LIN {X -0.028,Y -654.223,Z 1397.377,A 0.000,B 0.000,C 90.000,E1 103.772} C_DIS
LIN {X 0.258,Y -654.765,Z 1397.372,A 0.000,B 0.000,C 90.000,E1 103.008} C_DIS
LIN {X -0.090,Y -654.690,Z 1397.368,A 0.000,B 0.000,C 90.000,E1 102.299} C_DIS
LIN {X 0.196,Y -654.215,Z 1397.364,A 0.000,B 0.000,C 90.000,E1 101.535} C_DIS
LIN {X -0.172,Y -653.704,Z 1397.361,A 0.000,B 0.000,C 90.000,E1 101.074} C_DIS
LIN {X 0.100,Y -652.649,Z 1397.357,A 0.000,B 0.000,C 90.000,E1 100.310} C_DIS
LIN {X -0.269,Y -651.574,Z 1397.355,A 0.000,B 0.000,C 90.000,E1 99.849} C_DIS
LIN {X -0.133,Y -649.621,Z 1397.350,A 0.000,B 0.000,C 90.000,E1 99.095} C_DIS
LIN {X 0.226,Y -648.028,Z 1397.348,A 0.000,B 0.000,C 90.000,E1 98.568} C_DIS
LIN {X 0.320,Y -645.227,Z 1397.344,A 0.000,B 0.000,C 90.000,E1 97.814} C_DIS
LIN {X -0.334,Y -641.988,Z 1397.339,A 0.000,B 0.000,C 90.000,E1 97.125} C_DIS
LIN {X 0.006,Y -640.157,Z 1397.337,A 0.000,B 0.000,C 90.000,E1 96.720} C_DIS
LIN {X -0.120,Y -635.379,Z 1397.333,A 0.000,B 0.000,C 90.000,E1 95.853} C_DIS
LIN {X -0.229,Y -630.892,Z 1397.328,A 0.000,B 0.000,C 90.000,E1 95.106} C_DIS
LIN {X 0.039,Y -628.510,Z 1397.326,A 0.000,B 0.000,C 90.000,E1 94.702} C_DIS
LIN {X -0.040,Y -623.882,Z 1397.323,A 0.000,B 0.000,C 90.000,E1 94.073} C_DIS
LIN {X 0.039,Y -619.403,Z 1397.320,A 0.000,B 0.000,C 90.000,E1 93.555} C_DIS
LIN {X 0.122,Y -612.923,Z 1397.316,A 0.000,B 0.000,C 90.000,E1 92.922} C_DIS
LIN {X -0.217,Y -603.430,Z 1397.312,A 0.000,B 0.000,C 90.000,E1 92.121} C_DIS
LIN {X -0.253,Y -596.324,Z 1397.308,A 0.000,B 0.000,C 90.000,E1 91.547} C_DIS
LIN {X 0.108,Y -590.137,Z 1397.306,A 0.000,B 0.000,C 90.000,E1 91.088} C_DIS
LIN {X 0.184,Y -581.549,Z 1397.304,A 0.000,B 0.000,C 90.000,E1 90.630} C_DIS
LIN {X 0.247,Y -578.421,Z 1397.303,A 0.000,B 0.000,C 90.000,E1 90.458} C_DIS
LIN {X -0.091,Y -574.450,Z 1397.301,A 0.000,B 0.000,C 90.000,E1 90.172} C_DIS
LIN {X -0.127,Y -574.415,Z 1397.301,A 0.000,B 0.000,C 90.000,E1 90.172} C_DIS
LIN {X 0.227,Y -574.050,Z 1397.301,A 0.000,B 0.000,C 90.000,E1 90.057} C_DIS
LIN {X -0.012,Y -573.513,Z 1397.299,A 0.000,B 0.000,C 90.000,E1 89.828} C_DIS
LIN {X -0.202,Y -573.490,Z 1397.296,A 0.000,B 0.000,C 90.000,E1 89.370} C_DIS
LIN {X 0.249,Y -575.095,Z 1397.286,A 0.000,B 0.000,C 90.000,E1 87.421} C_DIS
LIN {X -0.237,Y -577.045,Z 1397.274,A 0.000,B 0.000,C 90.000,E1 85.298} C_DIS
LIN {X -0.145,Y -579.107,Z 1397.263,A 0.000,B 0.000,C 90.000,E1 83.394} C_DIS
LIN {X 0.007,Y -581.279,Z 1397.253,A 0.000,B 0.000,C 90.000,E1 81.489} C_DIS
LIN {X 0.257,Y -582.556,Z 1397.247,A 0.000,B 0.000,C 90.000,E1 80.387} C_DIS
LIN {X -0.052,Y -583.764,Z 1397.241,A 0.000,B 0.000,C 90.000,E1 79.342} C_DIS
LIN {X -0.236,Y -584.942,Z 1397.235,A 0.000,B 0.000,C 90.000,E1 78.285} C_DIS
LIN {X 0.094,Y -586.345,Z 1397.226,A 0.000,B 0.000,C 90.000,E1 76.645} C_DIS
LIN {X 0.019,Y -587.620,Z 1397.217,A 0.000,B 0.000,C 90.000,E1 75.046} C_DIS
LIN {X -0.040,Y -588.586,Z 1397.208,A 0.000,B 0.000,C 90.000,E1 73.449} C_DIS
LIN {X -0.063,Y -589.644,Z 1397.198,A 0.000,B 0.000,C 90.000,E1 71.583} C_DIS
LIN {X -0.302,Y -590.537,Z 1397.189,A 0.000,B 0.000,C 90.000,E1 70.007} C_DIS
LIN {X -0.097,Y -591.958,Z 1397.176,A 0.000,B 0.000,C 90.000,E1 67.592} C_DIS
LIN {X -0.192,Y -593.241,Z 1397.165,A 0.000,B 0.000,C 90.000,E1 65.741} C_DIS
LIN {X 0.124,Y -594.937,Z 1397.153,A 0.000,B 0.000,C 90.000,E1 63.589} C_DIS
LIN {X -0.049,Y -595.962,Z 1397.146,A 0.000,B 0.000,C 90.000,E1 62.281} C_DIS
LIN {X 0.329,Y -597.051,Z 1397.139,A 0.000,B 0.000,C 90.000,E1 60.923} C_DIS
LIN {X 0.281,Y -598.053,Z 1397.133,A 0.000,B 0.000,C 90.000,E1 59.871} C_DIS
LIN {X -0.130,Y -599.514,Z 1397.124,A 0.000,B 0.000,C 90.000,E1 58.329} C_DIS
LIN {X 0.074,Y -600.723,Z 1397.117,A 0.000,B 0.000,C 90.000,E1 56.993} C_DIS
LIN {X -0.126,Y -601.706,Z 1397.111,A 0.000,B 0.000,C 90.000,E1 55.960} C_DIS
LIN {X -0.049,Y -603.347,Z 1397.101,A 0.000,B 0.000,C 90.000,E1 54.116} C_DIS
LIN {X -0.187,Y -604.711,Z 1397.092,A 0.000,B 0.000,C 90.000,E1 52.557} C_DIS
LIN {X -0.201,Y -605.659,Z 1397.085,A 0.000,B 0.000,C 90.000,E1 51.251} C_DIS
LIN {X -0.084,Y -606.259,Z 1397.079,A 0.000,B 0.000,C 90.000,E1 50.194} C_DIS
LIN {X 0.047,Y -606.765,Z 1397.073,A 0.000,B 0.000,C 90.000,E1 49.138} C_DIS
LIN {X 0.250,Y -607.155,Z 1397.064,A 0.000,B 0.000,C 90.000,E1 47.553} C_DIS
LIN {X -0.255,Y -607.255,Z 1397.057,A 0.000,B 0.000,C 90.000,E1 46.296} C_DIS
LIN {X -0.337,Y -607.136,Z 1397.050,A 0.000,B 0.000,C 90.000,E1 45.000} C_DIS
LIN {X -0.230,Y -606.904,Z 1397.044,A 0.000,B 0.000,C 90.000,E1 43.947} C_DIS
LIN {X 0.117,Y -606.327,Z 1397.037,A 0.000,B 0.000,C 90.000,E1 42.609} C_DIS
LIN {X -0.211,Y -605.753,Z 1397.031,A 0.000,B 0.000,C 90.000,E1 41.595} C_DIS
LIN {X 0.165,Y -604.895,Z 1397.024,A 0.000,B 0.000,C 90.000,E1 40.253} C_DIS
LIN {X 0.013,Y -604.259,Z 1397.019,A 0.000,B 0.000,C 90.000,E1 39.483} C_DIS
LIN {X -0.019,Y -602.878,Z 1397.012,A 0.000,B 0.000,C 90.000,E1 38.177} C_DIS
LIN {X 0.269,Y -601.993,Z 1397.008,A 0.000,B 0.000,C 90.000,E1 37.363} C_DIS
LIN {X -0.164,Y -600.049,Z 1397.000,A 0.000,B 0.000,C 90.000,E1 36.091} C_DIS
LIN {X -0.270,Y -598.638,Z 1396.996,A 0.000,B 0.000,C 90.000,E1 35.311} C_DIS
LIN {X 0.101,Y -597.046,Z 1396.992,A 0.000,B 0.000,C 90.000,E1 34.485} C_DIS
LIN {X 0.077,Y -594.080,Z 1396.984,A 0.000,B 0.000,C 90.000,E1 33.166} C_DIS
LIN {X 0.395,Y -592.041,Z 1396.980,A 0.000,B 0.000,C 90.000,E1 32.339} C_DIS
LIN {X -0.240,Y -588.887,Z 1396.974,A 0.000,B 0.000,C 90.000,E1 31.337} C_DIS
LIN {X -0.167,Y -587.077,Z 1396.971,A 0.000,B 0.000,C 90.000,E1 30.797} C_DIS
LIN {X -0.231,Y -584.064,Z 1396.967,A 0.000,B 0.000,C 90.000,E1 30.001} C_DIS
LIN {X 0.179,Y -580.561,Z 1396.962,A 0.000,B 0.000,C 90.000,E1 29.155} C_DIS
LIN {X 0.187,Y -578.017,Z 1396.959,A 0.000,B 0.000,C 90.000,E1 28.615} C_DIS
LIN {X -0.180,Y -574.660,Z 1396.955,A 0.000,B 0.000,C 90.000,E1 27.975} C_DIS
LIN {X 0.120,Y -570.350,Z 1396.951,A 0.000,B 0.000,C 90.000,E1 27.129} C_DIS
LIN {X 0.114,Y -565.642,Z 1396.946,A 0.000,B 0.000,C 90.000,E1 26.309} C_DIS
LIN {X 0.305,Y -560.595,Z 1396.942,A 0.000,B 0.000,C 90.000,E1 25.463} C_DIS
LIN {X 0.303,Y -556.030,Z 1396.938,A 0.000,B 0.000,C 90.000,E1 24.771} C_DIS
LIN {X 0.146,Y -550.011,Z 1396.933,A 0.000,B 0.000,C 90.000,E1 23.951} C_DIS
LIN {X 0.049,Y -544.578,Z 1396.929,A 0.000,B 0.000,C 90.000,E1 23.259} C_DIS
LIN {X 0.060,Y -537.580,Z 1396.925,A 0.000,B 0.000,C 90.000,E1 22.408} C_DIS
LIN {X 0.026,Y -531.509,Z 1396.921,A 0.000,B 0.000,C 90.000,E1 21.716} C_DIS
LIN {X 0.295,Y -525.047,Z 1396.917,A 0.000,B 0.000,C 90.000,E1 20.972} C_DIS
LIN {X 0.144,Y -515.882,Z 1396.911,A 0.000,B 0.000,C 90.000,E1 19.993} C_DIS
LIN {X -0.024,Y -510.423,Z 1396.908,A 0.000,B 0.000,C 90.000,E1 19.450} C_DIS
LIN {X -0.067,Y -500.976,Z 1396.903,A 0.000,B 0.000,C 90.000,E1 18.489} C_DIS
LIN {X -0.077,Y -493.128,Z 1396.898,A 0.000,B 0.000,C 90.000,E1 17.692} C_DIS
LIN {X -0.209,Y -479.603,Z 1396.891,A 0.000,B 0.000,C 90.000,E1 16.315} C_DIS
LIN {X -0.202,Y -463.211,Z 1396.881,A 0.000,B 0.000,C 90.000,E1 14.592} C_DIS
LIN {X 0.213,Y -449.337,Z 1396.873,A 0.000,B 0.000,C 90.000,E1 13.063} C_DIS
LIN {X -0.042,Y -438.331,Z 1396.866,A 0.000,B 0.000,C 90.000,E1 11.883} C_DIS
LIN {X 0.139,Y -428.813,Z 1396.860,A 0.000,B 0.000,C 90.000,E1 10.782} C_DIS
LIN {X -0.148,Y -412.657,Z 1396.849,A 0.000,B 0.000,C 90.000,E1 8.859} C_DIS
LIN {X 0.054,Y -401.725,Z 1396.842,A 0.000,B 0.000,C 90.000,E1 7.466} C_DIS
LIN {X 0.139,Y -392.488,Z 1396.835,A 0.000,B 0.000,C 90.000,E1 6.258} C_DIS
LIN {X -0.029,Y -389.440,Z 1396.832,A 0.000,B 0.000,C 90.000,E1 5.796} C_DIS
LIN {X -0.162,Y -389.042,Z 1396.832,A 0.000,B 0.000,C 90.000,E1 5.682} C_DIS
LIN {X 0.188,Y -389.043,Z 1396.831,A 0.000,B 0.000,C 90.000,E1 5.625} C_DIS
LIN {X -0.051,Y -389.537,Z 1396.830,A 0.000,B 0.000,C 90.000,E1 5.454} C_DIS
LIN {X -0.089,Y -389.567,Z 1396.830,A 0.000,B 0.000,C 90.000,E1 5.454} C_DIS
LIN {X 0.043,Y -392.874,Z 1396.828,A 0.000,B 0.000,C 90.000,E1 5.049} C_DIS
LIN {X 0.057,Y -404.273,Z 1396.822,A 0.000,B 0.000,C 90.000,E1 4.012} C_DIS
LIN {X 0.016,Y -407.064,Z 1396.821,A 0.000,B 0.000,C 90.000,E1 3.726} C_DIS
LIN {X -0.104,Y -410.927,Z 1396.818,A 0.000,B 0.000,C 90.000,E1 3.326} C_DIS
LIN {X 0.192,Y -417.452,Z 1396.814,A 0.000,B 0.000,C 90.000,E1 2.465} C_DIS
LIN {X -0.142,Y -423.269,Z 1396.809,A 0.000,B 0.000,C 90.000,E1 1.661} C_DIS
LIN {X -0.021,Y -428.741,Z 1396.804,A 0.000,B 0.000,C 90.000,E1 0.802} C_DIS
LIN {X 0.000,Y -433.695,Z 1396.800,A 0.000,B 0.000,C 90.000,E1 360.000} C_DIS
LIN {X -0.029,Y -439.749,Z 1396.794,A 0.000,B 0.000,C 90.000,E1 358.969} C_DIS
LIN {X 0.200,Y -443.498,Z 1396.791,A 0.000,B 0.000,C 90.000,E1 358.282} C_DIS
LIN {X 0.100,Y -447.869,Z 1396.786,A 0.000,B 0.000,C 90.000,E1 357.478} C_DIS
LIN {X -0.032,Y -450.969,Z 1396.782,A 0.000,B 0.000,C 90.000,E1 356.846} C_DIS
LIN {X 0.205,Y -452.988,Z 1396.780,A 0.000,B 0.000,C 90.000,E1 356.331} C_DIS
LIN {X 0.029,Y -454.624,Z 1396.777,A 0.000,B 0.000,C 90.000,E1 355.869} C_DIS
LIN {X 0.196,Y -455.273,Z 1396.775,A 0.000,B 0.000,C 90.000,E1 355.527} C_DIS
LIN {X -0.088,Y -455.472,Z 1396.774,A 0.000,B 0.000,C 90.000,E1 355.241} C_DIS
LIN {X 0.121,Y -454.444,Z 1396.772,A 0.000,B 0.000,C 90.000,E1 354.894} C_DIS
LIN {X 0.092,Y -453.573,Z 1396.771,A 0.000,B 0.000,C 90.000,E1 354.837} C_DIS
LIN {X 0.144,Y -445.069,Z 1396.771,A 0.000,B 0.000,C 90.000,E1 354.723} C_DIS
LIN {X -0.018,Y -395.064,Z 1396.767,A 0.000,B 0.000,C 90.000,E1 354.090} C_DIS
LIN {X -0.030,Y -359.277,Z 1396.764,A 0.000,B 0.000,C 90.000,E1 353.514} C_DIS
LIN {X -0.057,Y -359.122,Z 1396.764,A 0.000,B 0.000,C 90.000,E1 353.514} C_DIS
LIN {X 0.002,Y -359.587,Z 1396.725,A 0.000,B 0.000,C 90.000,E1 346.520} C_DIS
LIN {X -0.087,Y -361.889,Z 1396.683,A 0.000,B 0.000,C 90.000,E1 339.028} C_DIS
LIN {X 0.160,Y -365.738,Z 1396.644,A 0.000,B 0.000,C 90.000,E1 331.897} C_DIS
LIN {X -0.082,Y -366.098,Z 1396.642,A 0.000,B 0.000,C 90.000,E1 331.563} C_DIS
LIN {X -0.039,Y -370.657,Z 1396.607,A 0.000,B 0.000,C 90.000,E1 325.261} C_DIS
LIN {X 0.006,Y -371.833,Z 1396.601,A 0.000,B 0.000,C 90.000,E1 324.149} C_DIS
LIN {X 0.023,Y -377.509,Z 1396.566,A 0.000,B 0.000,C 90.000,E1 317.919} C_DIS
LIN {X 0.035,Y -377.989,Z 1396.564,A 0.000,B 0.000,C 90.000,E1 317.553} C_DIS
LIN {X -0.202,Y -379.082,Z 1396.556,A 0.000,B 0.000,C 90.000,E1 316.134} C_DIS
LIN {X -0.194,Y -384.597,Z 1396.528,A 0.000,B 0.000,C 90.000,E1 311.067} C_DIS
LIN {X -0.149,Y -384.969,Z 1396.526,A 0.000,B 0.000,C 90.000,E1 310.701} C_DIS
LIN {X 0.020,Y -390.768,Z 1396.494,A 0.000,B 0.000,C 90.000,E1 304.945} C_DIS
LIN {X -0.136,Y -391.259,Z 1396.492,A 0.000,B 0.000,C 90.000,E1 304.612} C_DIS
LIN {X 0.019,Y -396.972,Z 1396.459,A 0.000,B 0.000,C 90.000,E1 298.565} C_DIS
LIN {X -0.031,Y -401.336,Z 1396.427,A 0.000,B 0.000,C 90.000,E1 292.950} C_DIS
LIN {X 0.050,Y -401.655,Z 1396.426,A 0.000,B 0.000,C 90.000,E1 292.589} C_DIS
LIN {X -0.185,Y -404.743,Z 1396.395,A 0.000,B 0.000,C 90.000,E1 287.040} C_DIS
LIN {X -0.182,Y -406.154,Z 1396.364,A 0.000,B 0.000,C 90.000,E1 281.478} C_DIS
LIN {X -0.084,Y -405.681,Z 1396.333,A 0.000,B 0.000,C 90.000,E1 275.910} C_DIS
LIN {X -0.012,Y -403.567,Z 1396.306,A 0.000,B 0.000,C 90.000,E1 271.031} C_DIS
LIN {X -0.077,Y -403.187,Z 1396.302,A 0.000,B 0.000,C 90.000,E1 270.344} C_DIS
LIN {X 0.156,Y -399.069,Z 1396.273,A 0.000,B 0.000,C 90.000,E1 265.065} C_DIS
LIN {X 0.097,Y -398.784,Z 1396.271,A 0.000,B 0.000,C 90.000,E1 264.723} C_DIS
LIN {X -0.013,Y -393.296,Z 1396.243,A 0.000,B 0.000,C 90.000,E1 259.803} C_DIS
LIN {X -0.093,Y -392.680,Z 1396.240,A 0.000,B 0.000,C 90.000,E1 259.106} C_DIS
LIN {X 0.079,Y -386.253,Z 1396.214,A 0.000,B 0.000,C 90.000,E1 254.448} C_DIS
LIN {X 0.043,Y -385.155,Z 1396.208,A 0.000,B 0.000,C 90.000,E1 253.378} C_DIS
LIN {X -0.200,Y -377.822,Z 1396.182,A 0.000,B 0.000,C 90.000,E1 248.720} C_DIS
LIN {X 0.022,Y -376.093,Z 1396.174,A 0.000,B 0.000,C 90.000,E1 247.230} C_DIS
LIN {X 0.080,Y -368.761,Z 1396.149,A 0.000,B 0.000,C 90.000,E1 242.820} C_DIS
LIN {X 0.064,Y -366.405,Z 1396.139,A 0.000,B 0.000,C 90.000,E1 240.973} C_DIS
LIN {X -0.087,Y -365.112,Z 1396.135,A 0.000,B 0.000,C 90.000,E1 240.255} C_DIS
LIN {X -0.021,Y -358.511,Z 1396.112,A 0.000,B 0.000,C 90.000,E1 236.135} C_DIS
LIN {X -0.170,Y -356.185,Z 1396.101,A 0.000,B 0.000,C 90.000,E1 234.276} C_DIS
LIN {X -0.022,Y -354.943,Z 1396.097,A 0.000,B 0.000,C 90.000,E1 233.497} C_DIS
LIN {X -0.039,Y -348.166,Z 1396.072,A 0.000,B 0.000,C 90.000,E1 228.933} C_DIS
LIN {X 0.131,Y -346.062,Z 1396.061,A 0.000,B 0.000,C 90.000,E1 226.986} C_DIS
LIN {X 0.012,Y -339.687,Z 1396.035,A 0.000,B 0.000,C 90.000,E1 222.366} C_DIS
LIN {X -0.175,Y -336.677,Z 1396.018,A 0.000,B 0.000,C 90.000,E1 219.277} C_DIS
LIN {X 0.195,Y -330.763,Z 1395.988,A 0.000,B 0.000,C 90.000,E1 213.706} C_DIS
LIN {X 0.147,Y -329.206,Z 1395.974,A 0.000,B 0.000,C 90.000,E1 211.337} C_DIS
LIN {X 0.043,Y -324.435,Z 1395.939,A 0.000,B 0.000,C 90.000,E1 204.975} C_DIS
LIN {X 0.165,Y -323.768,Z 1395.928,A 0.000,B 0.000,C 90.000,E1 202.950} C_DIS
LIN {X -0.045,Y -321.137,Z 1395.881,A 0.000,B 0.000,C 90.000,E1 194.537} C_DIS
LIN {X 0.122,Y -320.795,Z 1395.843,A 0.000,B 0.000,C 90.000,E1 187.757} C_DIS
LIN {X 0.104,Y -320.848,Z 1395.843,A 0.000,B 0.000,C 90.000,E1 187.757} C_DIS
LIN {X 0.026,Y -356.935,Z 1395.839,A 0.000,B 0.000,C 90.000,E1 187.004} C_DIS
LIN {X 0.156,Y -399.339,Z 1395.835,A 0.000,B 0.000,C 90.000,E1 186.258} C_DIS
LIN {X -0.126,Y -417.939,Z 1395.833,A 0.000,B 0.000,C 90.000,E1 186.024} C_DIS
LIN {X -0.135,Y -421.267,Z 1395.833,A 0.000,B 0.000,C 90.000,E1 185.967} C_DIS
LIN {X 0.206,Y -422.115,Z 1395.833,A 0.000,B 0.000,C 90.000,E1 185.853} C_DIS
LIN {X 0.014,Y -423.266,Z 1395.831,A 0.000,B 0.000,C 90.000,E1 185.625} C_DIS
LIN {X 0.086,Y -423.620,Z 1395.829,A 0.000,B 0.000,C 90.000,E1 185.277} C_DIS
LIN {X 0.123,Y -423.512,Z 1395.828,A 0.000,B 0.000,C 90.000,E1 184.935} C_DIS
LIN {X -0.076,Y -421.716,Z 1395.820,A 0.000,B 0.000,C 90.000,E1 183.612} C_DIS
LIN {X 0.059,Y -419.992,Z 1395.814,A 0.000,B 0.000,C 90.000,E1 182.579} C_DIS
LIN {X 0.125,Y -418.661,Z 1395.811,A 0.000,B 0.000,C 90.000,E1 181.892} C_DIS
LIN {X 0.194,Y -417.163,Z 1395.807,A 0.000,B 0.000,C 90.000,E1 181.203} C_DIS
LIN {X -0.158,Y -414.415,Z 1395.801,A 0.000,B 0.000,C 90.000,E1 180.229} C_DIS
LIN {X -0.131,Y -412.378,Z 1395.797,A 0.000,B 0.000,C 90.000,E1 179.542} C_DIS
LIN {X -0.125,Y -408.692,Z 1395.792,A 0.000,B 0.000,C 90.000,E1 178.511} C_DIS
LIN {X -0.148,Y -405.212,Z 1395.787,A 0.000,B 0.000,C 90.000,E1 177.650} C_DIS
LIN {X 0.201,Y -401.144,Z 1395.782,A 0.000,B 0.000,C 90.000,E1 176.731} C_DIS
LIN {X 0.076,Y -395.373,Z 1395.776,A 0.000,B 0.000,C 90.000,E1 175.698} C_DIS
LIN {X -0.133,Y -387.716,Z 1395.769,A 0.000,B 0.000,C 90.000,E1 174.489} C_DIS
LIN {X 0.002,Y -381.234,Z 1395.763,A 0.000,B 0.000,C 90.000,E1 173.394} C_DIS
LIN {X 0.114,Y -370.565,Z 1395.752,A 0.000,B 0.000,C 90.000,E1 171.376} C_DIS
LIN {X 0.179,Y -366.149,Z 1395.747,A 0.000,B 0.000,C 90.000,E1 170.443} C_DIS
LIN {X -0.111,Y -363.001,Z 1395.743,A 0.000,B 0.000,C 90.000,E1 169.746} C_DIS
LIN {X 0.015,Y -361.387,Z 1395.740,A 0.000,B 0.000,C 90.000,E1 169.218} C_DIS
LIN {X 0.117,Y -360.664,Z 1395.738,A 0.000,B 0.000,C 90.000,E1 168.814} C_DIS
LIN {X 0.080,Y -360.652,Z 1395.738,A 0.000,B 0.000,C 90.000,E1 168.814} C_DIS
LIN {X -0.165,Y -360.954,Z 1395.736,A 0.000,B 0.000,C 90.000,E1 168.578} C_DIS
LIN {X -0.023,Y -362.617,Z 1395.735,A 0.000,B 0.000,C 90.000,E1 168.229} C_DIS
LIN {X 0.071,Y -367.502,Z 1395.730,A 0.000,B 0.000,C 90.000,E1 167.465} C_DIS
LIN {X -0.133,Y -374.645,Z 1395.725,A 0.000,B 0.000,C 90.000,E1 166.589} C_DIS
LIN {X -0.073,Y -385.055,Z 1395.719,A 0.000,B 0.000,C 90.000,E1 165.408} C_DIS
LIN {X 0.174,Y -398.785,Z 1395.711,A 0.000,B 0.000,C 90.000,E1 163.976} C_DIS
LIN {X -0.061,Y -414.465,Z 1395.703,A 0.000,B 0.000,C 90.000,E1 162.598} C_DIS
LIN {X -0.047,Y -435.052,Z 1395.694,A 0.000,B 0.000,C 90.000,E1 160.913} C_DIS
LIN {X -0.120,Y -445.946,Z 1395.689,A 0.000,B 0.000,C 90.000,E1 160.061} C_DIS
LIN {X -0.065,Y -455.177,Z 1395.685,A 0.000,B 0.000,C 90.000,E1 159.316} C_DIS
LIN {X -0.197,Y -465.775,Z 1395.680,A 0.000,B 0.000,C 90.000,E1 158.465} C_DIS
LIN {X 0.082,Y -471.790,Z 1395.677,A 0.000,B 0.000,C 90.000,E1 157.922} C_DIS
LIN {X -0.062,Y -479.042,Z 1395.674,A 0.000,B 0.000,C 90.000,E1 157.283} C_DIS
LIN {X 0.206,Y -490.562,Z 1395.668,A 0.000,B 0.000,C 90.000,E1 156.177} C_DIS
LIN {X 0.033,Y -494.768,Z 1395.666,A 0.000,B 0.000,C 90.000,E1 155.793} C_DIS
LIN {X 0.115,Y -500.246,Z 1395.662,A 0.000,B 0.000,C 90.000,E1 155.229} C_DIS
LIN {X 0.091,Y -505.591,Z 1395.659,A 0.000,B 0.000,C 90.000,E1 154.665} C_DIS
LIN {X 0.111,Y -511.960,Z 1395.655,A 0.000,B 0.000,C 90.000,E1 153.948} C_DIS
LIN {X -0.026,Y -516.761,Z 1395.652,A 0.000,B 0.000,C 90.000,E1 153.384} C_DIS
LIN {X -0.170,Y -522.554,Z 1395.648,A 0.000,B 0.000,C 90.000,E1 152.666} C_DIS
LIN {X -0.098,Y -526.749,Z 1395.645,A 0.000,B 0.000,C 90.000,E1 152.076} C_DIS
LIN {X -0.250,Y -530.478,Z 1395.642,A 0.000,B 0.000,C 90.000,E1 151.513} C_DIS
LIN {X -0.124,Y -533.767,Z 1395.638,A 0.000,B 0.000,C 90.000,E1 150.923} C_DIS
LIN {X -0.115,Y -537.282,Z 1395.634,A 0.000,B 0.000,C 90.000,E1 150.205} C_DIS
LIN {X 0.196,Y -540.241,Z 1395.630,A 0.000,B 0.000,C 90.000,E1 149.459} C_DIS
LIN {X -0.072,Y -542.337,Z 1395.627,A 0.000,B 0.000,C 90.000,E1 148.918} C_DIS
LIN {X -0.129,Y -545.091,Z 1395.623,A 0.000,B 0.000,C 90.000,E1 148.074} C_DIS
LIN {X -0.073,Y -546.738,Z 1395.620,A 0.000,B 0.000,C 90.000,E1 147.502} C_DIS
LIN {X 0.204,Y -548.746,Z 1395.615,A 0.000,B 0.000,C 90.000,E1 146.628} C_DIS
LIN {X 0.043,Y -550.507,Z 1395.610,A 0.000,B 0.000,C 90.000,E1 145.801} C_DIS
LIN {X -0.160,Y -551.499,Z 1395.607,A 0.000,B 0.000,C 90.000,E1 145.261} C_DIS
LIN {X -0.041,Y -552.382,Z 1395.604,A 0.000,B 0.000,C 90.000,E1 144.689} C_DIS
LIN {X 0.153,Y -553.335,Z 1395.599,A 0.000,B 0.000,C 90.000,E1 143.829} C_DIS
LIN {X -0.272,Y -554.651,Z 1395.591,A 0.000,B 0.000,C 90.000,E1 142.477} C_DIS
LIN {X -0.265,Y -556.036,Z 1395.582,A 0.000,B 0.000,C 90.000,E1 140.803} C_DIS
LIN {X -0.035,Y -556.910,Z 1395.576,A 0.000,B 0.000,C 90.000,E1 139.666} C_DIS
LIN {X -0.053,Y -557.815,Z 1395.567,A 0.000,B 0.000,C 90.000,E1 138.000} C_DIS
LIN {X 0.311,Y -558.469,Z 1395.557,A 0.000,B 0.000,C 90.000,E1 136.296} C_DIS
LIN {X 0.216,Y -559.017,Z 1395.550,A 0.000,B 0.000,C 90.000,E1 134.919} C_DIS
LIN {X 0.127,Y -559.435,Z 1395.542,A 0.000,B 0.000,C 90.000,E1 133.542} C_DIS
LIN {X 0.069,Y -559.766,Z 1395.534,A 0.000,B 0.000,C 90.000,E1 132.162} C_DIS
LIN {X 0.221,Y -560.080,Z 1395.522,A 0.000,B 0.000,C 90.000,E1 129.930} C_DIS
LIN {X 0.084,Y -560.618,Z 1395.510,A 0.000,B 0.000,C 90.000,E1 127.729} C_DIS
LIN {X 0.063,Y -560.988,Z 1395.497,A 0.000,B 0.000,C 90.000,E1 125.518} C_DIS
LIN {X 0.028,Y -561.442,Z 1395.493,A 0.000,B 0.000,C 90.000,E1 124.692} C_DIS
LIN {X 0.013,Y -561.942,Z 1395.490,A 0.000,B 0.000,C 90.000,E1 124.278} C_DIS
LIN {X 0.078,Y -562.706,Z 1395.489,A 0.000,B 0.000,C 90.000,E1 123.992} C_DIS
LIN {X -0.035,Y -563.051,Z 1395.487,A 0.000,B 0.000,C 90.000,E1 123.706} C_DIS
LIN {X -0.077,Y -563.062,Z 1395.487,A 0.000,B 0.000,C 90.000,E1 123.706} C_DIS
LIN {X 0.172,Y -564.541,Z 1395.486,A 0.000,B 0.000,C 90.000,E1 123.499} C_DIS
LIN {X 0.146,Y -568.173,Z 1395.485,A 0.000,B 0.000,C 90.000,E1 123.372} C_DIS
LIN {X -0.107,Y -575.478,Z 1395.484,A 0.000,B 0.000,C 90.000,E1 123.214} C_DIS
LIN {X 0.122,Y -580.740,Z 1395.484,A 0.000,B 0.000,C 90.000,E1 123.086} C_DIS
LIN {X -0.122,Y -583.076,Z 1395.484,A 0.000,B 0.000,C 90.000,E1 123.038} C_DIS
LIN {X 0.264,Y -588.833,Z 1395.482,A 0.000,B 0.000,C 90.000,E1 122.752} C_DIS
LIN {X -0.072,Y -594.575,Z 1395.480,A 0.000,B 0.000,C 90.000,E1 122.467} C_DIS
LIN {X -0.332,Y -598.898,Z 1395.479,A 0.000,B 0.000,C 90.000,E1 122.212} C_DIS
LIN {X 0.131,Y -604.495,Z 1395.477,A 0.000,B 0.000,C 90.000,E1 121.750} C_DIS
LIN {X 0.023,Y -610.993,Z 1395.473,A 0.000,B 0.000,C 90.000,E1 121.180} C_DIS
LIN {X 0.203,Y -614.742,Z 1395.471,A 0.000,B 0.000,C 90.000,E1 120.797} C_DIS
LIN {X -0.275,Y -618.364,Z 1395.469,A 0.000,B 0.000,C 90.000,E1 120.463} C_DIS
LIN {X 0.050,Y -622.646,Z 1395.466,A 0.000,B 0.000,C 90.000,E1 119.922} C_DIS
LIN {X 0.053,Y -627.360,Z 1395.463,A 0.000,B 0.000,C 90.000,E1 119.283} C_DIS
LIN {X 0.088,Y -630.688,Z 1395.460,A 0.000,B 0.000,C 90.000,E1 118.771} C_DIS
LIN {X -0.091,Y -634.238,Z 1395.456,A 0.000,B 0.000,C 90.000,E1 118.153} C_DIS
LIN {X -0.011,Y -636.576,Z 1395.454,A 0.000,B 0.000,C 90.000,E1 117.641} C_DIS
LIN {X 0.034,Y -637.617,Z 1395.452,A 0.000,B 0.000,C 90.000,E1 117.385} C_DIS
LIN {X 0.195,Y -639.432,Z 1395.448,A 0.000,B 0.000,C 90.000,E1 116.616} C_DIS
LIN {X 0.313,Y -639.631,Z 1395.445,A 0.000,B 0.000,C 90.000,E1 116.104} C_DIS
LIN {X -0.202,Y -639.617,Z 1395.444,A 0.000,B 0.000,C 90.000,E1 115.899} C_DIS
LIN {X -0.358,Y -639.292,Z 1395.441,A 0.000,B 0.000,C 90.000,E1 115.412} C_DIS
LIN {X -0.298,Y -638.763,Z 1395.440,A 0.000,B 0.000,C 90.000,E1 115.155} C_DIS
LIN {X -0.239,Y -638.085,Z 1395.438,A 0.000,B 0.000,C 90.000,E1 114.899} C_DIS
LIN {X -0.182,Y -637.237,Z 1395.437,A 0.000,B 0.000,C 90.000,E1 114.643} C_DIS
LIN {X -0.083,Y -633.739,Z 1395.434,A 0.000,B 0.000,C 90.000,E1 114.131} C_DIS
LIN {X -0.062,Y -632.531,Z 1395.433,A 0.000,B 0.000,C 90.000,E1 114.003} C_DIS
LIN {X -0.123,Y -629.527,Z 1395.432,A 0.000,B 0.000,C 90.000,E1 113.770} C_DIS
LIN {X 0.316,Y -626.484,Z 1395.431,A 0.000,B 0.000,C 90.000,E1 113.515} C_DIS
LIN {X -0.241,Y -624.342,Z 1395.430,A 0.000,B 0.000,C 90.000,E1 113.462} C_DIS
LIN {X -0.278,Y -622.129,Z 1395.430,A 0.000,B 0.000,C 90.000,E1 113.387} C_DIS
LIN {X 0.254,Y -620.488,Z 1395.429,A 0.000,B 0.000,C 90.000,E1 113.259} C_DIS
LIN {X 0.116,Y -618.425,Z 1395.429,A 0.000,B 0.000,C 90.000,E1 113.153} C_DIS
LIN {X 0.088,Y -616.434,Z 1395.428,A 0.000,B 0.000,C 90.000,E1 113.078} C_DIS
LIN {X -0.181,Y -613.682,Z 1395.428,A 0.000,B 0.000,C 90.000,E1 113.025} C_DIS
LIN {X 0.300,Y -603.887,Z 1395.426,A 0.000,B 0.000,C 90.000,E1 112.642} C_DIS
LIN {X -0.172,Y -600.594,Z 1395.425,A 0.000,B 0.000,C 90.000,E1 112.589} C_DIS
LIN {X -0.210,Y -600.474,Z 1395.425,A 0.000,B 0.000,C 90.000,E1 112.589} C_DIS
LIN {X -0.194,Y -608.737,Z 1395.422,A 0.000,B 0.000,C 90.000,E1 111.950} C_DIS
LIN {X 0.170,Y -613.990,Z 1395.419,A 0.000,B 0.000,C 90.000,E1 111.482} C_DIS
LIN {X 0.002,Y -619.112,Z 1395.417,A 0.000,B 0.000,C 90.000,E1 111.046} C_DIS
LIN {X 0.131,Y -624.055,Z 1395.414,A 0.000,B 0.000,C 90.000,E1 110.556} C_DIS
LIN {X 0.053,Y -628.762,Z 1395.411,A 0.000,B 0.000,C 90.000,E1 110.066} C_DIS
LIN {X -0.128,Y -633.005,Z 1395.409,A 0.000,B 0.000,C 90.000,E1 109.577} C_DIS
LIN {X 0.305,Y -637.753,Z 1395.405,A 0.000,B 0.000,C 90.000,E1 108.906} C_DIS
LIN {X -0.012,Y -642.686,Z 1395.401,A 0.000,B 0.000,C 90.000,E1 108.181} C_DIS
LIN {X -0.287,Y -646.840,Z 1395.397,A 0.000,B 0.000,C 90.000,E1 107.457} C_DIS
LIN {X 0.231,Y -649.017,Z 1395.394,A 0.000,B 0.000,C 90.000,E1 106.913} C_DIS
LIN {X 0.091,Y -650.046,Z 1395.393,A 0.000,B 0.000,C 90.000,E1 106.677} C_DIS
LIN {X -0.178,Y -651.577,Z 1395.390,A 0.000,B 0.000,C 90.000,E1 106.205} C_DIS
LIN {X -0.128,Y -652.274,Z 1395.389,A 0.000,B 0.000,C 90.000,E1 105.953} C_DIS
LIN {X 0.125,Y -653.681,Z 1395.385,A 0.000,B 0.000,C 90.000,E1 105.190} C_DIS
LIN {X -0.349,Y -655.064,Z 1395.379,A 0.000,B 0.000,C 90.000,E1 104.245} C_DIS
LIN {X -0.054,Y -655.768,Z 1395.375,A 0.000,B 0.000,C 90.000,E1 103.480} C_DIS
LIN {X -0.279,Y -656.055,Z 1395.372,A 0.000,B 0.000,C 90.000,E1 103.008} C_DIS
LIN {X 0.026,Y -655.981,Z 1395.368,A 0.000,B 0.000,C 90.000,E1 102.243} C_DIS
LIN {X -0.201,Y -655.737,Z 1395.365,A 0.000,B 0.000,C 90.000,E1 101.771} C_DIS
LIN {X 0.211,Y -655.286,Z 1395.363,A 0.000,B 0.000,C 90.000,E1 101.243} C_DIS
LIN {X -0.149,Y -654.632,Z 1395.360,A 0.000,B 0.000,C 90.000,E1 100.782} C_DIS
LIN {X 0.130,Y -653.324,Z 1395.356,A 0.000,B 0.000,C 90.000,E1 100.018} C_DIS
LIN {X 0.278,Y -651.450,Z 1395.352,A 0.000,B 0.000,C 90.000,E1 99.265} C_DIS
LIN {X 0.144,Y -650.784,Z 1395.350,A 0.000,B 0.000,C 90.000,E1 99.029} C_DIS
LIN {X -0.232,Y -649.178,Z 1395.348,A 0.000,B 0.000,C 90.000,E1 98.568} C_DIS
LIN {X 0.025,Y -647.347,Z 1395.345,A 0.000,B 0.000,C 90.000,E1 98.049} C_DIS
LIN {X 0.115,Y -644.181,Z 1395.341,A 0.000,B 0.000,C 90.000,E1 97.296} C_DIS
LIN {X 0.216,Y -641.217,Z 1395.337,A 0.000,B 0.000,C 90.000,E1 96.663} C_DIS
LIN {X 0.231,Y -637.117,Z 1395.333,A 0.000,B 0.000,C 90.000,E1 95.910} C_DIS
LIN {X 0.135,Y -632.733,Z 1395.329,A 0.000,B 0.000,C 90.000,E1 95.163} C_DIS
LIN {X 0.275,Y -629.547,Z 1395.326,A 0.000,B 0.000,C 90.000,E1 94.645} C_DIS
LIN {X 0.248,Y -624.947,Z 1395.323,A 0.000,B 0.000,C 90.000,E1 94.012} C_DIS
LIN {X 0.289,Y -620.528,Z 1395.320,A 0.000,B 0.000,C 90.000,E1 93.498} C_DIS
LIN {X -0.258,Y -614.077,Z 1395.316,A 0.000,B 0.000,C 90.000,E1 92.922} C_DIS
LIN {X 0.023,Y -605.966,Z 1395.312,A 0.000,B 0.000,C 90.000,E1 92.178} C_DIS
LIN {X -0.040,Y -599.029,Z 1395.309,A 0.000,B 0.000,C 90.000,E1 91.604} C_DIS
LIN {X -0.025,Y -596.060,Z 1395.308,A 0.000,B 0.000,C 90.000,E1 91.375} C_DIS
LIN {X 0.223,Y -591.342,Z 1395.306,A 0.000,B 0.000,C 90.000,E1 91.031} C_DIS
LIN {X -0.251,Y -589.651,Z 1395.305,A 0.000,B 0.000,C 90.000,E1 90.974} C_DIS
LIN {X 0.020,Y -578.098,Z 1395.302,A 0.000,B 0.000,C 90.000,E1 90.344} C_DIS
LIN {X 0.013,Y -575.828,Z 1395.301,A 0.000,B 0.000,C 90.000,E1 90.172} C_DIS
LIN {X 0.005,Y -574.709,Z 1395.300,A 0.000,B 0.000,C 90.000,E1 90.057} C_DIS
LIN {X -0.104,Y -573.831,Z 1395.299,A 0.000,B 0.000,C 90.000,E1 89.885} C_DIS
LIN {X -0.063,Y -573.475,Z 1395.297,A 0.000,B 0.000,C 90.000,E1 89.542} C_DIS
LIN {X -0.260,Y -573.714,Z 1395.295,A 0.000,B 0.000,C 90.000,E1 89.026} C_DIS
LIN {X 0.048,Y -575.125,Z 1395.285,A 0.000,B 0.000,C 90.000,E1 87.364} C_DIS
LIN {X 0.099,Y -577.959,Z 1395.269,A 0.000,B 0.000,C 90.000,E1 84.375} C_DIS
LIN {X 0.225,Y -580.071,Z 1395.258,A 0.000,B 0.000,C 90.000,E1 82.470} C_DIS
LIN {X 0.256,Y -582.000,Z 1395.249,A 0.000,B 0.000,C 90.000,E1 80.849} C_DIS
LIN {X 0.181,Y -583.544,Z 1395.242,A 0.000,B 0.000,C 90.000,E1 79.511} C_DIS
LIN {X 0.125,Y -584.987,Z 1395.234,A 0.000,B 0.000,C 90.000,E1 78.173} C_DIS
LIN {X -0.120,Y -586.365,Z 1395.225,A 0.000,B 0.000,C 90.000,E1 76.589} C_DIS
LIN {X 0.120,Y -587.419,Z 1395.218,A 0.000,B 0.000,C 90.000,E1 75.227} C_DIS
LIN {X -0.116,Y -587.983,Z 1395.214,A 0.000,B 0.000,C 90.000,E1 74.448} C_DIS
LIN {X 0.151,Y -588.737,Z 1395.206,A 0.000,B 0.000,C 90.000,E1 73.087} C_DIS
LIN {X -0.106,Y -589.650,Z 1395.197,A 0.000,B 0.000,C 90.000,E1 71.511} C_DIS
LIN {X 0.221,Y -590.551,Z 1395.188,A 0.000,B 0.000,C 90.000,E1 69.880} C_DIS
LIN {X -0.233,Y -591.809,Z 1395.177,A 0.000,B 0.000,C 90.000,E1 67.794} C_DIS
LIN {X -0.199,Y -593.286,Z 1395.165,A 0.000,B 0.000,C 90.000,E1 65.665} C_DIS
LIN {X 0.220,Y -594.781,Z 1395.154,A 0.000,B 0.000,C 90.000,E1 63.768} C_DIS
LIN {X -0.226,Y -595.833,Z 1395.147,A 0.000,B 0.000,C 90.000,E1 62.487} C_DIS
LIN {X 0.092,Y -597.903,Z 1395.134,A 0.000,B 0.000,C 90.000,E1 60.078} C_DIS
LIN {X -0.098,Y -599.587,Z 1395.124,A 0.000,B 0.000,C 90.000,E1 58.250} C_DIS
LIN {X 0.111,Y -600.793,Z 1395.116,A 0.000,B 0.000,C 90.000,E1 56.914} C_DIS
LIN {X -0.085,Y -601.763,Z 1395.110,A 0.000,B 0.000,C 90.000,E1 55.881} C_DIS
LIN {X 0.233,Y -603.176,Z 1395.102,A 0.000,B 0.000,C 90.000,E1 54.276} C_DIS
LIN {X 0.086,Y -604.560,Z 1395.093,A 0.000,B 0.000,C 90.000,E1 52.718} C_DIS
LIN {X 0.064,Y -605.542,Z 1395.086,A 0.000,B 0.000,C 90.000,E1 51.412} C_DIS
LIN {X 0.176,Y -606.169,Z 1395.080,A 0.000,B 0.000,C 90.000,E1 50.356} C_DIS
LIN {X 0.304,Y -606.711,Z 1395.074,A 0.000,B 0.000,C 90.000,E1 49.299} C_DIS
LIN {X 0.054,Y -607.125,Z 1395.065,A 0.000,B 0.000,C 90.000,E1 47.757} C_DIS
LIN {X -0.004,Y -607.285,Z 1395.058,A 0.000,B 0.000,C 90.000,E1 46.458} C_DIS
LIN {X 0.102,Y -607.230,Z 1395.052,A 0.000,B 0.000,C 90.000,E1 45.405} C_DIS
LIN {X 0.021,Y -606.994,Z 1395.045,A 0.000,B 0.000,C 90.000,E1 44.109} C_DIS
LIN {X -0.072,Y -606.453,Z 1395.038,A 0.000,B 0.000,C 90.000,E1 42.813} C_DIS
LIN {X 0.048,Y -605.931,Z 1395.032,A 0.000,B 0.000,C 90.000,E1 41.757} C_DIS
LIN {X -0.033,Y -605.084,Z 1395.025,A 0.000,B 0.000,C 90.000,E1 40.458} C_DIS
LIN {X 0.073,Y -604.240,Z 1395.019,A 0.000,B 0.000,C 90.000,E1 39.402} C_DIS
LIN {X 0.039,Y -602.877,Z 1395.012,A 0.000,B 0.000,C 90.000,E1 38.096} C_DIS
LIN {X -0.267,Y -601.672,Z 1395.006,A 0.000,B 0.000,C 90.000,E1 37.076} C_DIS
LIN {X -0.111,Y -600.059,Z 1395.000,A 0.000,B 0.000,C 90.000,E1 36.011} C_DIS
LIN {X 0.020,Y -598.194,Z 1394.994,A 0.000,B 0.000,C 90.000,E1 34.945} C_DIS
LIN {X 0.008,Y -595.301,Z 1394.987,A 0.000,B 0.000,C 90.000,E1 33.627} C_DIS
LIN {X 0.015,Y -593.409,Z 1394.982,A 0.000,B 0.000,C 90.000,E1 32.832} C_DIS
LIN {X 0.327,Y -591.215,Z 1394.978,A 0.000,B 0.000,C 90.000,E1 32.005} C_DIS
LIN {X -0.201,Y -588.832,Z 1394.974,A 0.000,B 0.000,C 90.000,E1 31.258} C_DIS
LIN {X -0.131,Y -587.009,Z 1394.971,A 0.000,B 0.000,C 90.000,E1 30.718} C_DIS
LIN {X -0.199,Y -583.921,Z 1394.966,A 0.000,B 0.000,C 90.000,E1 29.922} C_DIS
LIN {X 0.273,Y -581.028,Z 1394.962,A 0.000,B 0.000,C 90.000,E1 29.205} C_DIS
LIN {X -0.140,Y -577.227,Z 1394.958,A 0.000,B 0.000,C 90.000,E1 28.437} C_DIS
LIN {X -0.237,Y -573.839,Z 1394.954,A 0.000,B 0.000,C 90.000,E1 27.769} C_DIS
LIN {X 0.049,Y -569.345,Z 1394.950,A 0.000,B 0.000,C 90.000,E1 26.924} C_DIS
LIN {X 0.031,Y -564.608,Z 1394.945,A 0.000,B 0.000,C 90.000,E1 26.104} C_DIS
LIN {X -0.032,Y -559.449,Z 1394.941,A 0.000,B 0.000,C 90.000,E1 25.283} C_DIS
LIN {X 0.065,Y -555.735,Z 1394.937,A 0.000,B 0.000,C 90.000,E1 24.719} C_DIS
LIN {X -0.089,Y -549.703,Z 1394.933,A 0.000,B 0.000,C 90.000,E1 23.898} C_DIS
LIN {X -0.184,Y -544.240,Z 1394.929,A 0.000,B 0.000,C 90.000,E1 23.206} C_DIS
LIN {X -0.196,Y -539.599,Z 1394.926,A 0.000,B 0.000,C 90.000,E1 22.642} C_DIS
LIN {X 0.254,Y -534.723,Z 1394.923,A 0.000,B 0.000,C 90.000,E1 22.025} C_DIS
LIN {X -0.285,Y -527.111,Z 1394.918,A 0.000,B 0.000,C 90.000,E1 21.227} C_DIS
LIN {X -0.262,Y -516.927,Z 1394.912,A 0.000,B 0.000,C 90.000,E1 20.120} C_DIS
LIN {X 0.093,Y -511.617,Z 1394.909,A 0.000,B 0.000,C 90.000,E1 19.523} C_DIS
LIN {X 0.101,Y -499.673,Z 1394.902,A 0.000,B 0.000,C 90.000,E1 18.308} C_DIS
LIN {X -0.166,Y -490.469,Z 1394.897,A 0.000,B 0.000,C 90.000,E1 17.402} C_DIS
LIN {X -0.001,Y -479.548,Z 1394.890,A 0.000,B 0.000,C 90.000,E1 16.260} C_DIS
LIN {X 0.139,Y -464.437,Z 1394.882,A 0.000,B 0.000,C 90.000,E1 14.662} C_DIS
LIN {X 0.103,Y -449.347,Z 1394.873,A 0.000,B 0.000,C 90.000,E1 13.063} C_DIS
LIN {X -0.126,Y -436.785,Z 1394.865,A 0.000,B 0.000,C 90.000,E1 11.715} C_DIS
LIN {X -0.094,Y -417.905,Z 1394.853,A 0.000,B 0.000,C 90.000,E1 9.500} C_DIS
LIN {X -0.206,Y -409.766,Z 1394.847,A 0.000,B 0.000,C 90.000,E1 8.511} C_DIS
LIN {X 0.138,Y -399.002,Z 1394.840,A 0.000,B 0.000,C 90.000,E1 7.125} C_DIS
LIN {X -0.127,Y -392.470,Z 1394.835,A 0.000,B 0.000,C 90.000,E1 6.315} C_DIS
LIN {X 0.094,Y -389.433,Z 1394.832,A 0.000,B 0.000,C 90.000,E1 5.796} C_DIS
LIN {X 0.152,Y -389.168,Z 1394.832,A 0.000,B 0.000,C 90.000,E1 5.682} C_DIS
LIN {X 0.113,Y -389.170,Z 1394.832,A 0.000,B 0.000,C 90.000,E1 5.682} C_DIS
LIN {X -0.172,Y -389.677,Z 1394.831,A 0.000,B 0.000,C 90.000,E1 5.568} C_DIS
LIN {X 0.178,Y -389.712,Z 1394.831,A 0.000,B 0.000,C 90.000,E1 5.511} C_DIS
LIN {X 0.171,Y -393.816,Z 1394.828,A 0.000,B 0.000,C 90.000,E1 5.049} C_DIS
LIN {X 0.097,Y -402.298,Z 1394.824,A 0.000,B 0.000,C 90.000,E1 4.302} C_DIS
LIN {X 0.165,Y -405.395,Z 1394.823,A 0.000,B 0.000,C 90.000,E1 4.012} C_DIS
LIN {X 0.013,Y -411.061,Z 1394.819,A 0.000,B 0.000,C 90.000,E1 3.440} C_DIS
LIN {X -0.079,Y -417.689,Z 1394.815,A 0.000,B 0.000,C 90.000,E1 2.636} C_DIS
LIN {X 0.041,Y -423.656,Z 1394.810,A 0.000,B 0.000,C 90.000,E1 1.776} C_DIS
LIN {X 0.198,Y -430.243,Z 1394.804,A 0.000,B 0.000,C 90.000,E1 0.745} C_DIS
LIN {X 0.000,Y -435.071,Z 1394.800,A 0.000,B 0.000,C 90.000,E1 360.000} C_DIS
LIN {X -0.072,Y -440.253,Z 1394.795,A 0.000,B 0.000,C 90.000,E1 359.141} C_DIS
LIN {X -0.218,Y -444.978,Z 1394.791,A 0.000,B 0.000,C 90.000,E1 358.339} C_DIS
LIN {X 0.140,Y -449.319,Z 1394.786,A 0.000,B 0.000,C 90.000,E1 357.478} C_DIS
LIN {X 0.102,Y -453.331,Z 1394.782,A 0.000,B 0.000,C 90.000,E1 356.674} C_DIS
LIN {X -0.017,Y -456.367,Z 1394.778,A 0.000,B 0.000,C 90.000,E1 356.045} C_DIS
LIN {X -0.175,Y -458.157,Z 1394.775,A 0.000,B 0.000,C 90.000,E1 355.584} C_DIS
LIN {X 0.004,Y -459.156,Z 1394.774,A 0.000,B 0.000,C 90.000,E1 355.241} C_DIS
LIN {X 0.227,Y -459.893,Z 1394.772,A 0.000,B 0.000,C 90.000,E1 354.894} C_DIS
LIN {X -0.046,Y -460.253,Z 1394.770,A 0.000,B 0.000,C 90.000,E1 354.609} C_DIS
LIN {X 0.186,Y -459.927,Z 1394.768,A 0.000,B 0.000,C 90.000,E1 354.261} C_DIS
LIN {X -0.230,Y -459.378,Z 1394.768,A 0.000,B 0.000,C 90.000,E1 354.204} C_DIS
LIN {X 0.062,Y -458.429,Z 1394.767,A 0.000,B 0.000,C 90.000,E1 354.090} C_DIS
LIN {X -0.010,Y -445.141,Z 1394.766,A 0.000,B 0.000,C 90.000,E1 353.913} C_DIS
LIN {X -0.193,Y -397.586,Z 1394.762,A 0.000,B 0.000,C 90.000,E1 353.223} C_DIS
LIN {X 0.040,Y -358.961,Z 1394.758,A 0.000,B 0.000,C 90.000,E1 352.470} C_DIS
LIN {X 0.010,Y -358.849,Z 1394.758,A 0.000,B 0.000,C 90.000,E1 352.470} C_DIS
LIN {X 0.033,Y -359.509,Z 1394.727,A 0.000,B 0.000,C 90.000,E1 346.756} C_DIS
LIN {X 0.116,Y -359.543,Z 1394.722,A 0.000,B 0.000,C 90.000,E1 345.992} C_DIS
LIN {X -0.128,Y -361.965,Z 1394.683,A 0.000,B 0.000,C 90.000,E1 338.901} C_DIS
LIN {X -0.114,Y -366.194,Z 1394.641,A 0.000,B 0.000,C 90.000,E1 331.435} C_DIS
LIN {X -0.089,Y -371.219,Z 1394.604,A 0.000,B 0.000,C 90.000,E1 324.769} C_DIS
LIN {X -0.102,Y -371.652,Z 1394.602,A 0.000,B 0.000,C 90.000,E1 324.402} C_DIS
LIN {X -0.045,Y -376.756,Z 1394.570,A 0.000,B 0.000,C 90.000,E1 318.528} C_DIS
LIN {X 0.244,Y -378.150,Z 1394.564,A 0.000,B 0.000,C 90.000,E1 317.391} C_DIS
LIN {X -0.016,Y -384.275,Z 1394.529,A 0.000,B 0.000,C 90.000,E1 311.272} C_DIS
LIN {X 0.025,Y -384.778,Z 1394.527,A 0.000,B 0.000,C 90.000,E1 310.906} C_DIS
LIN {X 0.015,Y -390.945,Z 1394.494,A 0.000,B 0.000,C 90.000,E1 304.818} C_DIS
LIN {X -0.139,Y -391.363,Z 1394.492,A 0.000,B 0.000,C 90.000,E1 304.485} C_DIS
LIN {X 0.031,Y -397.071,Z 1394.458,A 0.000,B 0.000,C 90.000,E1 298.437} C_DIS
LIN {X -0.013,Y -401.479,Z 1394.427,A 0.000,B 0.000,C 90.000,E1 292.823} C_DIS
LIN {X -0.219,Y -401.766,Z 1394.423,A 0.000,B 0.000,C 90.000,E1 292.153} C_DIS
LIN {X 0.114,Y -404.560,Z 1394.396,A 0.000,B 0.000,C 90.000,E1 287.221} C_DIS
LIN {X -0.173,Y -404.761,Z 1394.394,A 0.000,B 0.000,C 90.000,E1 286.913} C_DIS
LIN {X 0.121,Y -406.035,Z 1394.365,A 0.000,B 0.000,C 90.000,E1 281.658} C_DIS
LIN {X 0.211,Y -406.141,Z 1394.363,A 0.000,B 0.000,C 90.000,E1 281.299} C_DIS
LIN {X -0.162,Y -405.654,Z 1394.334,A 0.000,B 0.000,C 90.000,E1 276.144} C_DIS
LIN {X -0.157,Y -405.606,Z 1394.332,A 0.000,B 0.000,C 90.000,E1 275.796} C_DIS
LIN {X -0.084,Y -403.550,Z 1394.305,A 0.000,B 0.000,C 90.000,E1 270.917} C_DIS
LIN {X -0.149,Y -403.048,Z 1394.301,A 0.000,B 0.000,C 90.000,E1 270.229} C_DIS
LIN {X 0.076,Y -399.013,Z 1394.272,A 0.000,B 0.000,C 90.000,E1 264.951} C_DIS
LIN {X -0.030,Y -397.641,Z 1394.266,A 0.000,B 0.000,C 90.000,E1 263.913} C_DIS
LIN {X -0.150,Y -392.928,Z 1394.241,A 0.000,B 0.000,C 90.000,E1 259.342} C_DIS
LIN {X -0.157,Y -391.880,Z 1394.237,A 0.000,B 0.000,C 90.000,E1 258.634} C_DIS
LIN {X -0.019,Y -385.739,Z 1394.211,A 0.000,B 0.000,C 90.000,E1 253.976} C_DIS
LIN {X -0.083,Y -384.978,Z 1394.207,A 0.000,B 0.000,C 90.000,E1 253.268} C_DIS
LIN {X 0.144,Y -378.122,Z 1394.183,A 0.000,B 0.000,C 90.000,E1 248.901} C_DIS
LIN {X -0.120,Y -376.362,Z 1394.175,A 0.000,B 0.000,C 90.000,E1 247.486} C_DIS
LIN {X 0.005,Y -375.866,Z 1394.173,A 0.000,B 0.000,C 90.000,E1 247.102} C_DIS
LIN {X -0.044,Y -369.092,Z 1394.150,A 0.000,B 0.000,C 90.000,E1 243.076} C_DIS
LIN {X 0.034,Y -366.245,Z 1394.138,A 0.000,B 0.000,C 90.000,E1 240.845} C_DIS
LIN {X -0.004,Y -358.840,Z 1394.113,A 0.000,B 0.000,C 90.000,E1 236.373} C_DIS
LIN {X -0.016,Y -356.030,Z 1394.101,A 0.000,B 0.000,C 90.000,E1 234.116} C_DIS
LIN {X -0.019,Y -348.468,Z 1394.073,A 0.000,B 0.000,C 90.000,E1 229.175} C_DIS
LIN {X 0.042,Y -345.885,Z 1394.060,A 0.000,B 0.000,C 90.000,E1 226.863} C_DIS
LIN {X 0.009,Y -339.113,Z 1394.032,A 0.000,B 0.000,C 90.000,E1 221.838} C_DIS
LIN {X 0.092,Y -336.950,Z 1394.020,A 0.000,B 0.000,C 90.000,E1 219.483} C_DIS
LIN {X 0.073,Y -331.626,Z 1393.993,A 0.000,B 0.000,C 90.000,E1 214.771} C_DIS
LIN {X 0.144,Y -329.365,Z 1393.976,A 0.000,B 0.000,C 90.000,E1 211.592} C_DIS
LIN {X 0.155,Y -328.638,Z 1393.971,A 0.000,B 0.000,C 90.000,E1 210.797} C_DIS
LIN {X 0.068,Y -324.090,Z 1393.934,A 0.000,B 0.000,C 90.000,E1 204.027} C_DIS
LIN {X -0.123,Y -323.868,Z 1393.929,A 0.000,B 0.000,C 90.000,E1 203.259} C_DIS
LIN {X 0.050,Y -323.111,Z 1393.922,A 0.000,B 0.000,C 90.000,E1 202.025} C_DIS
LIN {X 0.159,Y -321.122,Z 1393.880,A 0.000,B 0.000,C 90.000,E1 194.356} C_DIS
LIN {X 0.066,Y -320.536,Z 1393.850,A 0.000,B 0.000,C 90.000,E1 188.916} C_DIS
LIN {X 0.047,Y -320.652,Z 1393.850,A 0.000,B 0.000,C 90.000,E1 188.916} C_DIS
LIN {X -0.090,Y -354.494,Z 1393.845,A 0.000,B 0.000,C 90.000,E1 188.106} C_DIS
LIN {X 0.089,Y -393.343,Z 1393.841,A 0.000,B 0.000,C 90.000,E1 187.296} C_DIS
LIN {X 0.023,Y -421.073,Z 1393.838,A 0.000,B 0.000,C 90.000,E1 186.834} C_DIS
LIN {X -0.023,Y -424.271,Z 1393.838,A 0.000,B 0.000,C 90.000,E1 186.777} C_DIS
LIN {X -0.153,Y -425.146,Z 1393.837,A 0.000,B 0.000,C 90.000,E1 186.720} C_DIS
LIN {X 0.039,Y -426.314,Z 1393.836,A 0.000,B 0.000,C 90.000,E1 186.429} C_DIS
LIN {X 0.079,Y -426.794,Z 1393.834,A 0.000,B 0.000,C 90.000,E1 186.087} C_DIS
LIN {X 0.169,Y -426.791,Z 1393.832,A 0.000,B 0.000,C 90.000,E1 185.739} C_DIS
LIN {X -0.165,Y -426.551,Z 1393.830,A 0.000,B 0.000,C 90.000,E1 185.448} C_DIS
LIN {X 0.022,Y -425.392,Z 1393.825,A 0.000,B 0.000,C 90.000,E1 184.416} C_DIS
LIN {X 0.201,Y -423.978,Z 1393.819,A 0.000,B 0.000,C 90.000,E1 183.383} C_DIS
LIN {X -0.059,Y -422.306,Z 1393.813,A 0.000,B 0.000,C 90.000,E1 182.407} C_DIS
LIN {X 0.040,Y -421.026,Z 1393.810,A 0.000,B 0.000,C 90.000,E1 181.718} C_DIS
LIN {X 0.116,Y -419.578,Z 1393.806,A 0.000,B 0.000,C 90.000,E1 181.031} C_DIS
LIN {X 0.181,Y -417.830,Z 1393.802,A 0.000,B 0.000,C 90.000,E1 180.344} C_DIS
LIN {X -0.162,Y -414.855,Z 1393.796,A 0.000,B 0.000,C 90.000,E1 179.370} C_DIS
LIN {X -0.126,Y -411.170,Z 1393.791,A 0.000,B 0.000,C 90.000,E1 178.339} C_DIS
LIN {X -0.118,Y -408.470,Z 1393.787,A 0.000,B 0.000,C 90.000,E1 177.650} C_DIS
LIN {X -0.139,Y -404.589,Z 1393.782,A 0.000,B 0.000,C 90.000,E1 176.788} C_DIS
LIN {X 0.178,Y -398.851,Z 1393.776,A 0.000,B 0.000,C 90.000,E1 175.698} C_DIS
LIN {X 0.018,Y -392.379,Z 1393.770,A 0.000,B 0.000,C 90.000,E1 174.666} C_DIS
LIN {X -0.126,Y -386.770,Z 1393.766,A 0.000,B 0.000,C 90.000,E1 173.799} C_DIS
LIN {X 0.058,Y -381.547,Z 1393.760,A 0.000,B 0.000,C 90.000,E1 172.875} C_DIS
LIN {X 0.108,Y -375.599,Z 1393.755,A 0.000,B 0.000,C 90.000,E1 171.781} C_DIS
LIN {X 0.007,Y -368.180,Z 1393.746,A 0.000,B 0.000,C 90.000,E1 170.330} C_DIS
LIN {X 0.107,Y -364.339,Z 1393.741,A 0.000,B 0.000,C 90.000,E1 169.398} C_DIS
LIN {X -0.043,Y -363.178,Z 1393.739,A 0.000,B 0.000,C 90.000,E1 169.050} C_DIS
LIN {X 0.130,Y -362.372,Z 1393.737,A 0.000,B 0.000,C 90.000,E1 168.578} C_DIS
LIN {X 0.135,Y -362.313,Z 1393.736,A 0.000,B 0.000,C 90.000,E1 168.522} C_DIS
LIN {X 0.099,Y -362.313,Z 1393.736,A 0.000,B 0.000,C 90.000,E1 168.522} C_DIS
LIN {X -0.178,Y -363.932,Z 1393.734,A 0.000,B 0.000,C 90.000,E1 168.173} C_DIS
LIN {X 0.135,Y -364.535,Z 1393.733,A 0.000,B 0.000,C 90.000,E1 167.937} C_DIS
LIN {X 0.200,Y -367.558,Z 1393.731,A 0.000,B 0.000,C 90.000,E1 167.465} C_DIS
LIN {X -0.070,Y -374.684,Z 1393.725,A 0.000,B 0.000,C 90.000,E1 166.589} C_DIS
LIN {X 0.036,Y -383.367,Z 1393.720,A 0.000,B 0.000,C 90.000,E1 165.574} C_DIS
LIN {X -0.082,Y -395.475,Z 1393.713,A 0.000,B 0.000,C 90.000,E1 164.338} C_DIS
LIN {X -0.232,Y -409.110,Z 1393.706,A 0.000,B 0.000,C 90.000,E1 163.087} C_DIS
LIN {X -0.003,Y -432.633,Z 1393.695,A 0.000,B 0.000,C 90.000,E1 161.094} C_DIS
LIN {X -0.163,Y -443.710,Z 1393.690,A 0.000,B 0.000,C 90.000,E1 160.242} C_DIS
LIN {X 0.125,Y -454.640,Z 1393.685,A 0.000,B 0.000,C 90.000,E1 159.337} C_DIS
LIN {X 0.120,Y -465.407,Z 1393.681,A 0.000,B 0.000,C 90.000,E1 158.465} C_DIS
LIN {X -0.009,Y -472.828,Z 1393.677,A 0.000,B 0.000,C 90.000,E1 157.847} C_DIS
LIN {X 0.152,Y -478.620,Z 1393.674,A 0.000,B 0.000,C 90.000,E1 157.305} C_DIS
LIN {X 0.189,Y -490.120,Z 1393.668,A 0.000,B 0.000,C 90.000,E1 156.230} C_DIS
LIN {X -0.057,Y -495.693,Z 1393.665,A 0.000,B 0.000,C 90.000,E1 155.717} C_DIS
LIN {X 0.221,Y -503.859,Z 1393.660,A 0.000,B 0.000,C 90.000,E1 154.845} C_DIS
LIN {X -0.018,Y -510.321,Z 1393.656,A 0.000,B 0.000,C 90.000,E1 154.152} C_DIS
LIN {X -0.047,Y -515.329,Z 1393.653,A 0.000,B 0.000,C 90.000,E1 153.563} C_DIS
LIN {X 0.099,Y -522.329,Z 1393.648,A 0.000,B 0.000,C 90.000,E1 152.666} C_DIS
LIN {X -0.080,Y -526.592,Z 1393.645,A 0.000,B 0.000,C 90.000,E1 152.103} C_DIS
LIN {X 0.017,Y -530.334,Z 1393.642,A 0.000,B 0.000,C 90.000,E1 151.513} C_DIS
LIN {X -0.003,Y -534.359,Z 1393.638,A 0.000,B 0.000,C 90.000,E1 150.795} C_DIS
LIN {X 0.153,Y -537.194,Z 1393.635,A 0.000,B 0.000,C 90.000,E1 150.205} C_DIS
LIN {X -0.276,Y -540.170,Z 1393.631,A 0.000,B 0.000,C 90.000,E1 149.537} C_DIS
LIN {X -0.084,Y -542.272,Z 1393.627,A 0.000,B 0.000,C 90.000,E1 148.948} C_DIS
LIN {X 0.140,Y -545.039,Z 1393.623,A 0.000,B 0.000,C 90.000,E1 148.074} C_DIS
LIN {X -0.097,Y -546.699,Z 1393.620,A 0.000,B 0.000,C 90.000,E1 147.533} C_DIS
LIN {X -0.285,Y -548.684,Z 1393.615,A 0.000,B 0.000,C 90.000,E1 146.707} C_DIS
LIN {X 0.314,Y -550.452,Z 1393.610,A 0.000,B 0.000,C 90.000,E1 145.801} C_DIS
LIN {X 0.110,Y -551.453,Z 1393.607,A 0.000,B 0.000,C 90.000,E1 145.261} C_DIS
LIN {X 0.228,Y -552.322,Z 1393.604,A 0.000,B 0.000,C 90.000,E1 144.689} C_DIS
LIN {X 0.096,Y -553.282,Z 1393.599,A 0.000,B 0.000,C 90.000,E1 143.863} C_DIS
LIN {X -0.003,Y -554.578,Z 1393.592,A 0.000,B 0.000,C 90.000,E1 142.477} C_DIS
LIN {X 0.077,Y -556.169,Z 1393.581,A 0.000,B 0.000,C 90.000,E1 140.517} C_DIS
LIN {X 0.309,Y -556.975,Z 1393.575,A 0.000,B 0.000,C 90.000,E1 139.380} C_DIS
LIN {X -0.129,Y -557.842,Z 1393.565,A 0.000,B 0.000,C 90.000,E1 137.757} C_DIS
LIN {X -0.036,Y -558.697,Z 1393.553,A 0.000,B 0.000,C 90.000,E1 135.526} C_DIS
LIN {X 0.265,Y -559.150,Z 1393.545,A 0.000,B 0.000,C 90.000,E1 134.109} C_DIS
LIN {X -0.209,Y -559.584,Z 1393.538,A 0.000,B 0.000,C 90.000,E1 132.771} C_DIS
LIN {X 0.075,Y -559.734,Z 1393.531,A 0.000,B 0.000,C 90.000,E1 131.634} C_DIS
LIN {X -0.133,Y -560.139,Z 1393.519,A 0.000,B 0.000,C 90.000,E1 129.439} C_DIS
LIN {X 0.338,Y -560.540,Z 1393.510,A 0.000,B 0.000,C 90.000,E1 127.729} C_DIS
LIN {X 0.088,Y -561.281,Z 1393.496,A 0.000,B 0.000,C 90.000,E1 125.264} C_DIS
LIN {X -0.066,Y -561.572,Z 1393.494,A 0.000,B 0.000,C 90.000,E1 124.865} C_DIS
LIN {X -0.087,Y -562.364,Z 1393.491,A 0.000,B 0.000,C 90.000,E1 124.405} C_DIS
LIN {X 0.115,Y -564.007,Z 1393.489,A 0.000,B 0.000,C 90.000,E1 124.040} C_DIS
LIN {X 0.072,Y -564.169,Z 1393.489,A 0.000,B 0.000,C 90.000,E1 123.992} C_DIS
LIN {X 0.030,Y -564.204,Z 1393.489,A 0.000,B 0.000,C 90.000,E1 123.992} C_DIS
LIN {X 0.080,Y -565.552,Z 1393.489,A 0.000,B 0.000,C 90.000,E1 123.913} C_DIS
LIN {X 0.120,Y -569.195,Z 1393.488,A 0.000,B 0.000,C 90.000,E1 123.785} C_DIS
LIN {X 0.299,Y -571.546,Z 1393.487,A 0.000,B 0.000,C 90.000,E1 123.706} C_DIS
LIN {X -0.032,Y -576.250,Z 1393.487,A 0.000,B 0.000,C 90.000,E1 123.658} C_DIS
LIN {X 0.137,Y -579.198,Z 1393.487,A 0.000,B 0.000,C 90.000,E1 123.579} C_DIS
LIN {X -0.148,Y -585.338,Z 1393.486,A 0.000,B 0.000,C 90.000,E1 123.420} C_DIS
LIN {X -0.264,Y -590.798,Z 1393.484,A 0.000,B 0.000,C 90.000,E1 123.166} C_DIS
LIN {X -0.119,Y -596.572,Z 1393.482,A 0.000,B 0.000,C 90.000,E1 122.801} C_DIS
LIN {X -0.278,Y -602.294,Z 1393.480,A 0.000,B 0.000,C 90.000,E1 122.418} C_DIS
LIN {X -0.200,Y -606.419,Z 1393.478,A 0.000,B 0.000,C 90.000,E1 122.084} C_DIS
LIN {X 0.072,Y -611.694,Z 1393.476,A 0.000,B 0.000,C 90.000,E1 121.592} C_DIS
LIN {X -0.241,Y -615.441,Z 1393.474,A 0.000,B 0.000,C 90.000,E1 121.258} C_DIS
LIN {X 0.115,Y -620.179,Z 1393.471,A 0.000,B 0.000,C 90.000,E1 120.718} C_DIS
LIN {X 0.092,Y -624.487,Z 1393.468,A 0.000,B 0.000,C 90.000,E1 120.207} C_DIS
LIN {X -0.131,Y -628.377,Z 1393.465,A 0.000,B 0.000,C 90.000,E1 119.716} C_DIS
LIN {X -0.082,Y -632.623,Z 1393.462,A 0.000,B 0.000,C 90.000,E1 119.077} C_DIS
LIN {X -0.012,Y -635.603,Z 1393.459,A 0.000,B 0.000,C 90.000,E1 118.565} C_DIS
LIN {X 0.108,Y -638.749,Z 1393.455,A 0.000,B 0.000,C 90.000,E1 117.924} C_DIS
LIN {X -0.048,Y -640.569,Z 1393.452,A 0.000,B 0.000,C 90.000,E1 117.436} C_DIS
LIN {X 0.012,Y -641.398,Z 1393.451,A 0.000,B 0.000,C 90.000,E1 117.180} C_DIS
LIN {X 0.074,Y -641.955,Z 1393.450,A 0.000,B 0.000,C 90.000,E1 116.924} C_DIS
LIN {X -0.078,Y -642.498,Z 1393.447,A 0.000,B 0.000,C 90.000,E1 116.437} C_DIS
LIN {X 0.065,Y -642.599,Z 1393.444,A 0.000,B 0.000,C 90.000,E1 115.924} C_DIS
LIN {X 0.137,Y -642.508,Z 1393.443,A 0.000,B 0.000,C 90.000,E1 115.668} C_DIS
LIN {X 0.278,Y -641.837,Z 1393.440,A 0.000,B 0.000,C 90.000,E1 115.155} C_DIS
LIN {X -0.138,Y -639.755,Z 1393.437,A 0.000,B 0.000,C 90.000,E1 114.567} C_DIS
LIN {X -0.284,Y -636.312,Z 1393.434,A 0.000,B 0.000,C 90.000,E1 114.079} C_DIS
LIN {X -0.257,Y -635.260,Z 1393.433,A 0.000,B 0.000,C 90.000,E1 113.951} C_DIS
LIN {X 0.157,Y -628.991,Z 1393.430,A 0.000,B 0.000,C 90.000,E1 113.462} C_DIS
LIN {X -0.152,Y -627.021,Z 1393.430,A 0.000,B 0.000,C 90.000,E1 113.387} C_DIS
LIN {X -0.032,Y -621.279,Z 1393.429,A 0.000,B 0.000,C 90.000,E1 113.131} C_DIS
LIN {X -0.209,Y -619.920,Z 1393.428,A 0.000,B 0.000,C 90.000,E1 113.078} C_DIS
LIN {X -0.297,Y -614.056,Z 1393.427,A 0.000,B 0.000,C 90.000,E1 112.898} C_DIS
LIN {X 0.179,Y -603.509,Z 1393.425,A 0.000,B 0.000,C 90.000,E1 112.514} C_DIS
LIN {X 0.142,Y -603.426,Z 1393.425,A 0.000,B 0.000,C 90.000,E1 112.514} C_DIS
LIN {X 0.000,Y -607.241,Z 1393.423,A 0.000,B 0.000,C 90.000,E1 112.206} C_DIS
LIN {X -0.314,Y -613.656,Z 1393.421,A 0.000,B 0.000,C 90.000,E1 111.716} C_DIS
LIN {X 0.038,Y -618.844,Z 1393.418,A 0.000,B 0.000,C 90.000,E1 111.227} C_DIS
LIN {X 0.178,Y -623.857,Z 1393.415,A 0.000,B 0.000,C 90.000,E1 110.737} C_DIS
LIN {X 0.076,Y -628.634,Z 1393.413,A 0.000,B 0.000,C 90.000,E1 110.248} C_DIS
LIN {X -0.116,Y -633.944,Z 1393.409,A 0.000,B 0.000,C 90.000,E1 109.631} C_DIS
LIN {X 0.325,Y -638.633,Z 1393.406,A 0.000,B 0.000,C 90.000,E1 108.960} C_DIS
LIN {X -0.006,Y -642.809,Z 1393.402,A 0.000,B 0.000,C 90.000,E1 108.362} C_DIS
LIN {X -0.126,Y -645.742,Z 1393.399,A 0.000,B 0.000,C 90.000,E1 107.873} C_DIS
LIN {X 0.193,Y -648.363,Z 1393.396,A 0.000,B 0.000,C 90.000,E1 107.347} C_DIS
LIN {X 0.105,Y -650.501,Z 1393.394,A 0.000,B 0.000,C 90.000,E1 106.858} C_DIS
LIN {X -0.030,Y -651.524,Z 1393.392,A 0.000,B 0.000,C 90.000,E1 106.622} C_DIS
LIN {X -0.233,Y -653.665,Z 1393.388,A 0.000,B 0.000,C 90.000,E1 105.898} C_DIS
LIN {X 0.036,Y -655.035,Z 1393.384,A 0.000,B 0.000,C 90.000,E1 105.134} C_DIS
LIN {X -0.256,Y -656.457,Z 1393.379,A 0.000,B 0.000,C 90.000,E1 104.175} C_DIS
LIN {X 0.045,Y -657.097,Z 1393.375,A 0.000,B 0.000,C 90.000,E1 103.411} C_DIS
LIN {X -0.174,Y -657.338,Z 1393.372,A 0.000,B 0.000,C 90.000,E1 102.939} C_DIS
LIN {X 0.247,Y -657.363,Z 1393.369,A 0.000,B 0.000,C 90.000,E1 102.411} C_DIS
LIN {X -0.219,Y -656.988,Z 1393.365,A 0.000,B 0.000,C 90.000,E1 101.715} C_DIS
LIN {X 0.202,Y -656.501,Z 1393.362,A 0.000,B 0.000,C 90.000,E1 101.186} C_DIS
LIN {X -0.027,Y -655.835,Z 1393.360,A 0.000,B 0.000,C 90.000,E1 100.715} C_DIS
LIN {X 0.144,Y -654.426,Z 1393.355,A 0.000,B 0.000,C 90.000,E1 99.962} C_DIS
LIN {X 0.304,Y -652.546,Z 1393.351,A 0.000,B 0.000,C 90.000,E1 99.208} C_DIS
LIN {X -0.060,Y -651.041,Z 1393.349,A 0.000,B 0.000,C 90.000,E1 98.746} C_DIS
LIN {X 0.307,Y -649.348,Z 1393.346,A 0.000,B 0.000,C 90.000,E1 98.219} C_DIS
LIN {X 0.071,Y -648.438,Z 1393.344,A 0.000,B 0.000,C 90.000,E1 97.992} C_DIS
LIN {X 0.171,Y -645.181,Z 1393.340,A 0.000,B 0.000,C 90.000,E1 97.239} C_DIS
LIN {X 0.283,Y -642.176,Z 1393.337,A 0.000,B 0.000,C 90.000,E1 96.606} C_DIS
LIN {X -0.200,Y -638.781,Z 1393.333,A 0.000,B 0.000,C 90.000,E1 96.024} C_DIS
LIN {X -0.278,Y -634.453,Z 1393.329,A 0.000,B 0.000,C 90.000,E1 95.277} C_DIS
LIN {X -0.261,Y -630.461,Z 1393.326,A 0.000,B 0.000,C 90.000,E1 94.645} C_DIS
LIN {X -0.180,Y -626.889,Z 1393.323,A 0.000,B 0.000,C 90.000,E1 94.131} C_DIS
LIN {X -0.078,Y -622.637,Z 1393.320,A 0.000,B 0.000,C 90.000,E1 93.612} C_DIS
LIN {X 0.252,Y -620.215,Z 1393.319,A 0.000,B 0.000,C 90.000,E1 93.326} C_DIS
LIN {X -0.174,Y -615.052,Z 1393.316,A 0.000,B 0.000,C 90.000,E1 92.865} C_DIS
LIN {X 0.261,Y -608.486,Z 1393.313,A 0.000,B 0.000,C 90.000,E1 92.236} C_DIS
LIN {X 0.134,Y -601.612,Z 1393.309,A 0.000,B 0.000,C 90.000,E1 91.661} C_DIS
LIN {X 0.136,Y -597.281,Z 1393.307,A 0.000,B 0.000,C 90.000,E1 91.318} C_DIS
LIN {X 0.182,Y -594.064,Z 1393.306,A 0.000,B 0.000,C 90.000,E1 91.088} C_DIS
LIN {X 0.052,Y -589.169,Z 1393.305,A 0.000,B 0.000,C 90.000,E1 90.802} C_DIS
LIN {X -0.090,Y -577.706,Z 1393.301,A 0.000,B 0.000,C 90.000,E1 90.229} C_DIS
LIN {X 0.225,Y -576.623,Z 1393.301,A 0.000,B 0.000,C 90.000,E1 90.115} C_DIS
LIN {X 0.266,Y -574.495,Z 1393.300,A 0.000,B 0.000,C 90.000,E1 89.885} C_DIS
LIN {X -0.174,Y -573.998,Z 1393.299,A 0.000,B 0.000,C 90.000,E1 89.828} C_DIS
LIN {X -0.231,Y -573.523,Z 1393.297,A 0.000,B 0.000,C 90.000,E1 89.427} C_DIS
LIN {X 0.043,Y -573.953,Z 1393.293,A 0.000,B 0.000,C 90.000,E1 88.682} C_DIS
LIN {X 0.209,Y -575.125,Z 1393.285,A 0.000,B 0.000,C 90.000,E1 87.306} C_DIS
LIN {X -0.172,Y -578.255,Z 1393.267,A 0.000,B 0.000,C 90.000,E1 84.090} C_DIS
LIN {X -0.050,Y -580.398,Z 1393.257,A 0.000,B 0.000,C 90.000,E1 82.186} C_DIS
LIN {X -0.162,Y -582.013,Z 1393.249,A 0.000,B 0.000,C 90.000,E1 80.849} C_DIS
LIN {X -0.238,Y -583.564,Z 1393.242,A 0.000,B 0.000,C 90.000,E1 79.511} C_DIS
LIN {X -0.295,Y -584.996,Z 1393.234,A 0.000,B 0.000,C 90.000,E1 78.173} C_DIS
LIN {X 0.029,Y -586.358,Z 1393.225,A 0.000,B 0.000,C 90.000,E1 76.533} C_DIS
LIN {X 0.019,Y -587.233,Z 1393.219,A 0.000,B 0.000,C 90.000,E1 75.463} C_DIS
LIN {X 0.029,Y -588.001,Z 1393.213,A 0.000,B 0.000,C 90.000,E1 74.393} C_DIS
LIN {X 0.144,Y -588.857,Z 1393.204,A 0.000,B 0.000,C 90.000,E1 72.779} C_DIS
LIN {X 0.030,Y -589.636,Z 1393.197,A 0.000,B 0.000,C 90.000,E1 71.456} C_DIS
LIN {X -0.203,Y -590.552,Z 1393.188,A 0.000,B 0.000,C 90.000,E1 69.880} C_DIS
LIN {X 0.115,Y -591.808,Z 1393.176,A 0.000,B 0.000,C 90.000,E1 67.720} C_DIS
LIN {X -0.083,Y -593.310,Z 1393.165,A 0.000,B 0.000,C 90.000,E1 65.613} C_DIS
LIN {X -0.206,Y -594.815,Z 1393.154,A 0.000,B 0.000,C 90.000,E1 63.768} C_DIS
LIN {X -0.034,Y -595.679,Z 1393.148,A 0.000,B 0.000,C 90.000,E1 62.692} C_DIS
LIN {X -0.036,Y -597.940,Z 1393.134,A 0.000,B 0.000,C 90.000,E1 60.049} C_DIS
LIN {X -0.016,Y -599.626,Z 1393.123,A 0.000,B 0.000,C 90.000,E1 58.201} C_DIS
LIN {X -0.076,Y -601.081,Z 1393.115,A 0.000,B 0.000,C 90.000,E1 56.628} C_DIS
LIN {X 0.324,Y -601.794,Z 1393.110,A 0.000,B 0.000,C 90.000,E1 55.801} C_DIS
LIN {X -0.195,Y -603.215,Z 1393.101,A 0.000,B 0.000,C 90.000,E1 54.276} C_DIS
LIN {X 0.025,Y -604.593,Z 1393.093,A 0.000,B 0.000,C 90.000,E1 52.683} C_DIS
LIN {X 0.278,Y -605.728,Z 1393.084,A 0.000,B 0.000,C 90.000,E1 51.090} C_DIS
LIN {X 0.011,Y -606.313,Z 1393.078,A 0.000,B 0.000,C 90.000,E1 50.070} C_DIS
LIN {X -0.124,Y -606.725,Z 1393.074,A 0.000,B 0.000,C 90.000,E1 49.299} C_DIS
LIN {X 0.075,Y -607.145,Z 1393.065,A 0.000,B 0.000,C 90.000,E1 47.715} C_DIS
LIN {X -0.013,Y -607.330,Z 1393.058,A 0.000,B 0.000,C 90.000,E1 46.419} C_DIS
LIN {X -0.082,Y -607.240,Z 1393.051,A 0.000,B 0.000,C 90.000,E1 45.121} C_DIS
LIN {X 0.265,Y -606.915,Z 1393.043,A 0.000,B 0.000,C 90.000,E1 43.785} C_DIS
LIN {X -0.246,Y -606.352,Z 1393.036,A 0.000,B 0.000,C 90.000,E1 42.528} C_DIS
LIN {X -0.120,Y -605.762,Z 1393.030,A 0.000,B 0.000,C 90.000,E1 41.472} C_DIS
LIN {X -0.198,Y -604.893,Z 1393.023,A 0.000,B 0.000,C 90.000,E1 40.172} C_DIS
LIN {X -0.093,Y -604.026,Z 1393.017,A 0.000,B 0.000,C 90.000,E1 39.116} C_DIS
LIN {X -0.128,Y -602.627,Z 1393.010,A 0.000,B 0.000,C 90.000,E1 37.810} C_DIS
LIN {X 0.154,Y -601.749,Z 1393.006,A 0.000,B 0.000,C 90.000,E1 36.996} C_DIS
LIN {X 0.203,Y -599.710,Z 1392.998,A 0.000,B 0.000,C 90.000,E1 35.678} C_DIS
LIN {X 0.094,Y -598.289,Z 1392.994,A 0.000,B 0.000,C 90.000,E1 34.898} C_DIS
LIN {X 0.314,Y -594.767,Z 1392.985,A 0.000,B 0.000,C 90.000,E1 33.293} C_DIS
LIN {X -0.181,Y -592.793,Z 1392.981,A 0.000,B 0.000,C 90.000,E1 32.546} C_DIS
LIN {X 0.008,Y -589.692,Z 1392.975,A 0.000,B 0.000,C 90.000,E1 31.465} C_DIS
LIN {X 0.086,Y -587.965,Z 1392.972,A 0.000,B 0.000,C 90.000,E1 30.924} C_DIS
LIN {X 0.149,Y -586.052,Z 1392.969,A 0.000,B 0.000,C 90.000,E1 30.384} C_DIS
LIN {X 0.068,Y -582.802,Z 1392.964,A 0.000,B 0.000,C 90.000,E1 29.589} C_DIS
LIN {X -0.193,Y -580.421,Z 1392.961,A 0.000,B 0.000,C 90.000,E1 29.077} C_DIS
LIN {X 0.100,Y -575.961,Z 1392.956,A 0.000,B 0.000,C 90.000,E1 28.103} C_DIS
LIN {X -0.201,Y -573.147,Z 1392.953,A 0.000,B 0.000,C 90.000,E1 27.590} C_DIS
LIN {X -0.003,Y -567.778,Z 1392.948,A 0.000,B 0.000,C 90.000,E1 26.616} C_DIS
LIN {X 0.058,Y -563.770,Z 1392.944,A 0.000,B 0.000,C 90.000,E1 25.924} C_DIS
LIN {X 0.328,Y -559.435,Z 1392.940,A 0.000,B 0.000,C 90.000,E1 25.207} C_DIS
LIN {X -0.084,Y -555.705,Z 1392.937,A 0.000,B 0.000,C 90.000,E1 24.695} C_DIS
LIN {X 0.258,Y -549.666,Z 1392.932,A 0.000,B 0.000,C 90.000,E1 23.823} C_DIS
LIN {X -0.058,Y -544.197,Z 1392.929,A 0.000,B 0.000,C 90.000,E1 23.153} C_DIS
LIN {X -0.069,Y -539.550,Z 1392.926,A 0.000,B 0.000,C 90.000,E1 22.589} C_DIS
LIN {X 0.240,Y -533.381,Z 1392.922,A 0.000,B 0.000,C 90.000,E1 21.844} C_DIS
LIN {X -0.291,Y -525.715,Z 1392.917,A 0.000,B 0.000,C 90.000,E1 21.046} C_DIS
LIN {X 0.182,Y -515.420,Z 1392.911,A 0.000,B 0.000,C 90.000,E1 19.885} C_DIS
LIN {X -0.168,Y -511.393,Z 1392.908,A 0.000,B 0.000,C 90.000,E1 19.504} C_DIS
LIN {X 0.020,Y -500.948,Z 1392.902,A 0.000,B 0.000,C 90.000,E1 18.417} C_DIS
LIN {X 0.087,Y -490.332,Z 1392.896,A 0.000,B 0.000,C 90.000,E1 17.330} C_DIS
LIN {X 0.052,Y -479.309,Z 1392.890,A 0.000,B 0.000,C 90.000,E1 16.205} C_DIS
LIN {X -0.028,Y -465.500,Z 1392.882,A 0.000,B 0.000,C 90.000,E1 14.773} C_DIS
LIN {X -0.189,Y -450.184,Z 1392.873,A 0.000,B 0.000,C 90.000,E1 13.175} C_DIS
LIN {X -0.021,Y -434.869,Z 1392.864,A 0.000,B 0.000,C 90.000,E1 11.478} C_DIS
LIN {X -0.188,Y -414.512,Z 1392.850,A 0.000,B 0.000,C 90.000,E1 9.095} C_DIS
LIN {X 0.089,Y -406.311,Z 1392.845,A 0.000,B 0.000,C 90.000,E1 8.049} C_DIS
LIN {X -0.170,Y -392.685,Z 1392.835,A 0.000,B 0.000,C 90.000,E1 6.372} C_DIS
LIN {X -0.088,Y -389.505,Z 1392.833,A 0.000,B 0.000,C 90.000,E1 5.853} C_DIS
LIN {X 0.084,Y -389.282,Z 1392.832,A 0.000,B 0.000,C 90.000,E1 5.739} C_DIS
LIN {X 0.046,Y -389.281,Z 1392.832,A 0.000,B 0.000,C 90.000,E1 5.739} C_DIS
LIN {X -0.135,Y -389.553,Z 1392.832,A 0.000,B 0.000,C 90.000,E1 5.682} C_DIS
LIN {X -0.173,Y -389.573,Z 1392.831,A 0.000,B 0.000,C 90.000,E1 5.682} C_DIS
LIN {X 0.091,Y -393.170,Z 1392.829,A 0.000,B 0.000,C 90.000,E1 5.220} C_DIS
LIN {X 0.007,Y -403.066,Z 1392.824,A 0.000,B 0.000,C 90.000,E1 4.359} C_DIS
LIN {X -0.133,Y -407.663,Z 1392.822,A 0.000,B 0.000,C 90.000,E1 3.955} C_DIS
LIN {X -0.100,Y -411.902,Z 1392.819,A 0.000,B 0.000,C 90.000,E1 3.498} C_DIS
LIN {X -0.036,Y -418.003,Z 1392.815,A 0.000,B 0.000,C 90.000,E1 2.751} C_DIS
LIN {X 0.048,Y -424.928,Z 1392.810,A 0.000,B 0.000,C 90.000,E1 1.776} C_DIS
LIN {X -0.212,Y -431.555,Z 1392.804,A 0.000,B 0.000,C 90.000,E1 0.802} C_DIS
LIN {X 0.000,Y -436.446,Z 1392.800,A 0.000,B 0.000,C 90.000,E1 360.000} C_DIS
LIN {X -0.060,Y -441.698,Z 1392.795,A 0.000,B 0.000,C 90.000,E1 359.141} C_DIS
LIN {X -0.193,Y -446.458,Z 1392.791,A 0.000,B 0.000,C 90.000,E1 358.339} C_DIS
LIN {X 0.181,Y -450.775,Z 1392.786,A 0.000,B 0.000,C 90.000,E1 357.478} C_DIS
LIN {X 0.072,Y -454.078,Z 1392.783,A 0.000,B 0.000,C 90.000,E1 356.846} C_DIS
LIN {X 0.051,Y -457.922,Z 1392.778,A 0.000,B 0.000,C 90.000,E1 356.045} C_DIS
LIN {X 0.090,Y -461.331,Z 1392.774,A 0.000,B 0.000,C 90.000,E1 355.241} C_DIS
LIN {X 0.059,Y -463.507,Z 1392.770,A 0.000,B 0.000,C 90.000,E1 354.609} C_DIS
LIN {X -0.159,Y -464.271,Z 1392.768,A 0.000,B 0.000,C 90.000,E1 354.318} C_DIS
LIN {X 0.092,Y -464.763,Z 1392.767,A 0.000,B 0.000,C 90.000,E1 353.970} C_DIS
LIN {X -0.167,Y -464.753,Z 1392.765,A 0.000,B 0.000,C 90.000,E1 353.685} C_DIS
LIN {X -0.065,Y -464.333,Z 1392.764,A 0.000,B 0.000,C 90.000,E1 353.514} C_DIS
LIN {X 0.089,Y -462.822,Z 1392.763,A 0.000,B 0.000,C 90.000,E1 353.337} C_DIS
LIN {X -0.040,Y -405.151,Z 1392.758,A 0.000,B 0.000,C 90.000,E1 352.413} C_DIS
LIN {X -0.059,Y -367.866,Z 1392.754,A 0.000,B 0.000,C 90.000,E1 351.659} C_DIS
LIN {X 0.074,Y -358.887,Z 1392.753,A 0.000,B 0.000,C 90.000,E1 351.432} C_DIS
LIN {X 0.040,Y -358.698,Z 1392.752,A 0.000,B 0.000,C 90.000,E1 351.432} C_DIS
LIN {X -0.083,Y -359.586,Z 1392.725,A 0.000,B 0.000,C 90.000,E1 346.520} C_DIS
LIN {X -0.171,Y -361.898,Z 1392.683,A 0.000,B 0.000,C 90.000,E1 339.028} C_DIS
LIN {X 0.075,Y -365.750,Z 1392.644,A 0.000,B 0.000,C 90.000,E1 331.897} C_DIS
LIN {X 0.155,Y -366.111,Z 1392.642,A 0.000,B 0.000,C 90.000,E1 331.513} C_DIS
LIN {X -0.124,Y -370.671,Z 1392.607,A 0.000,B 0.000,C 90.000,E1 325.261} C_DIS
LIN {X 0.148,Y -371.511,Z 1392.603,A 0.000,B 0.000,C 90.000,E1 324.482} C_DIS
LIN {X -0.089,Y -372.046,Z 1392.599,A 0.000,B 0.000,C 90.000,E1 323.783} C_DIS
LIN {X -0.050,Y -378.006,Z 1392.564,A 0.000,B 0.000,C 90.000,E1 317.553} C_DIS
LIN {X 0.001,Y -379.688,Z 1392.552,A 0.000,B 0.000,C 90.000,E1 315.364} C_DIS
LIN {X 0.008,Y -384.615,Z 1392.528,A 0.000,B 0.000,C 90.000,E1 311.024} C_DIS
LIN {X 0.060,Y -385.221,Z 1392.524,A 0.000,B 0.000,C 90.000,E1 310.297} C_DIS
LIN {X -0.223,Y -391.273,Z 1392.492,A 0.000,B 0.000,C 90.000,E1 304.612} C_DIS
LIN {X -0.070,Y -396.986,Z 1392.459,A 0.000,B 0.000,C 90.000,E1 298.565} C_DIS
LIN {X -0.118,Y -401.351,Z 1392.427,A 0.000,B 0.000,C 90.000,E1 292.950} C_DIS
LIN {X -0.038,Y -401.658,Z 1392.426,A 0.000,B 0.000,C 90.000,E1 292.589} C_DIS
LIN {X 0.114,Y -404.748,Z 1392.395,A 0.000,B 0.000,C 90.000,E1 286.985} C_DIS
LIN {X 0.128,Y -406.157,Z 1392.364,A 0.000,B 0.000,C 90.000,E1 281.422} C_DIS
LIN {X -0.172,Y -405.676,Z 1392.333,A 0.000,B 0.000,C 90.000,E1 275.910} C_DIS
LIN {X -0.100,Y -403.565,Z 1392.306,A 0.000,B 0.000,C 90.000,E1 271.031} C_DIS
LIN {X -0.165,Y -403.172,Z 1392.302,A 0.000,B 0.000,C 90.000,E1 270.344} C_DIS
LIN {X 0.068,Y -399.064,Z 1392.273,A 0.000,B 0.000,C 90.000,E1 265.065} C_DIS
LIN {X 0.010,Y -398.765,Z 1392.271,A 0.000,B 0.000,C 90.000,E1 264.723} C_DIS
LIN {X -0.101,Y -393.286,Z 1392.243,A 0.000,B 0.000,C 90.000,E1 259.803} C_DIS
LIN {X -0.179,Y -392.658,Z 1392.239,A 0.000,B 0.000,C 90.000,E1 259.106} C_DIS
LIN {X -0.008,Y -386.239,Z 1392.214,A 0.000,B 0.000,C 90.000,E1 254.448} C_DIS
LIN {X -0.043,Y -385.141,Z 1392.208,A 0.000,B 0.000,C 90.000,E1 253.378} C_DIS
LIN {X 0.066,Y -377.806,Z 1392.182,A 0.000,B 0.000,C 90.000,E1 248.666} C_DIS
LIN {X -0.063,Y -376.074,Z 1392.173,A 0.000,B 0.000,C 90.000,E1 247.230} C_DIS
LIN {X -0.006,Y -368.742,Z 1392.149,A 0.000,B 0.000,C 90.000,E1 242.820} C_DIS
LIN {X -0.021,Y -366.389,Z 1392.139,A 0.000,B 0.000,C 90.000,E1 240.973} C_DIS
LIN {X 0.145,Y -365.087,Z 1392.135,A 0.000,B 0.000,C 90.000,E1 240.205} C_DIS
LIN {X -0.105,Y -358.493,Z 1392.112,A 0.000,B 0.000,C 90.000,E1 236.135} C_DIS
LIN {X -0.046,Y -356.170,Z 1392.101,A 0.000,B 0.000,C 90.000,E1 234.242} C_DIS
LIN {X -0.107,Y -354.919,Z 1392.097,A 0.000,B 0.000,C 90.000,E1 233.497} C_DIS
LIN {X -0.122,Y -348.150,Z 1392.072,A 0.000,B 0.000,C 90.000,E1 228.933} C_DIS
LIN {X 0.048,Y -346.048,Z 1392.061,A 0.000,B 0.000,C 90.000,E1 226.986} C_DIS
LIN {X 0.020,Y -339.247,Z 1392.033,A 0.000,B 0.000,C 90.000,E1 221.962} C_DIS
LIN {X -0.115,Y -337.051,Z 1392.020,A 0.000,B 0.000,C 90.000,E1 219.644} C_DIS
LIN {X 0.217,Y -336.657,Z 1392.018,A 0.000,B 0.000,C 90.000,E1 219.197} C_DIS
LIN {X 0.113,Y -330.751,Z 1391.987,A 0.000,B 0.000,C 90.000,E1 213.706} C_DIS
LIN {X 0.065,Y -329.192,Z 1391.974,A 0.000,B 0.000,C 90.000,E1 211.337} C_DIS
LIN {X 0.100,Y -324.429,Z 1391.939,A 0.000,B 0.000,C 90.000,E1 204.951} C_DIS
LIN {X 0.084,Y -323.757,Z 1391.928,A 0.000,B 0.000,C 90.000,E1 202.950} C_DIS
LIN {X -0.126,Y -321.139,Z 1391.881,A 0.000,B 0.000,C 90.000,E1 194.537} C_DIS
LIN {X 0.028,Y -320.410,Z 1391.856,A 0.000,B 0.000,C 90.000,E1 190.074} C_DIS
LIN {X 0.010,Y -320.506,Z 1391.856,A 0.000,B 0.000,C 90.000,E1 190.074} C_DIS
LIN {X 0.132,Y -350.579,Z 1391.851,A 0.000,B 0.000,C 90.000,E1 189.208} C_DIS
LIN {X -0.070,Y -386.553,Z 1391.847,A 0.000,B 0.000,C 90.000,E1 188.398} C_DIS
LIN {X 0.154,Y -426.747,Z 1391.842,A 0.000,B 0.000,C 90.000,E1 187.587} C_DIS
LIN {X 0.048,Y -427.772,Z 1391.842,A 0.000,B 0.000,C 90.000,E1 187.530} C_DIS
LIN {X 0.104,Y -428.955,Z 1391.841,A 0.000,B 0.000,C 90.000,E1 187.296} C_DIS
LIN {X 0.203,Y -429.555,Z 1391.839,A 0.000,B 0.000,C 90.000,E1 186.947} C_DIS
LIN {X -0.171,Y -429.661,Z 1391.837,A 0.000,B 0.000,C 90.000,E1 186.663} C_DIS
LIN {X 0.038,Y -429.327,Z 1391.833,A 0.000,B 0.000,C 90.000,E1 185.967} C_DIS
LIN {X 0.198,Y -428.860,Z 1391.829,A 0.000,B 0.000,C 90.000,E1 185.277} C_DIS
LIN {X -0.011,Y -427.726,Z 1391.824,A 0.000,B 0.000,C 90.000,E1 184.302} C_DIS
LIN {X 0.198,Y -426.395,Z 1391.818,A 0.000,B 0.000,C 90.000,E1 183.269} C_DIS
LIN {X -0.034,Y -424.826,Z 1391.813,A 0.000,B 0.000,C 90.000,E1 182.293} C_DIS
LIN {X 0.085,Y -423.548,Z 1391.809,A 0.000,B 0.000,C 90.000,E1 181.604} C_DIS
LIN {X 0.134,Y -422.878,Z 1391.807,A 0.000,B 0.000,C 90.000,E1 181.260} C_DIS
LIN {X -0.153,Y -420.469,Z 1391.802,A 0.000,B 0.000,C 90.000,E1 180.286} C_DIS
LIN {X -0.079,Y -418.652,Z 1391.798,A 0.000,B 0.000,C 90.000,E1 179.599} C_DIS
LIN {X -0.019,Y -416.437,Z 1391.794,A 0.000,B 0.000,C 90.000,E1 178.912} C_DIS
LIN {X 0.021,Y -414.001,Z 1391.790,A 0.000,B 0.000,C 90.000,E1 178.224} C_DIS
LIN {X 0.048,Y -412.111,Z 1391.787,A 0.000,B 0.000,C 90.000,E1 177.707} C_DIS
LIN {X 0.063,Y -408.339,Z 1391.783,A 0.000,B 0.000,C 90.000,E1 176.846} C_DIS
LIN {X 0.027,Y -404.763,Z 1391.779,A 0.000,B 0.000,C 90.000,E1 176.159} C_DIS
LIN {X -0.012,Y -400.861,Z 1391.775,A 0.000,B 0.000,C 90.000,E1 175.469} C_DIS
LIN {X -0.082,Y -396.604,Z 1391.771,A 0.000,B 0.000,C 90.000,E1 174.780} C_DIS
LIN {X 0.107,Y -387.533,Z 1391.763,A 0.000,B 0.000,C 90.000,E1 173.337} C_DIS
LIN {X 0.073,Y -378.252,Z 1391.754,A 0.000,B 0.000,C 90.000,E1 171.724} C_DIS
LIN {X -0.013,Y -369.890,Z 1391.745,A 0.000,B 0.000,C 90.000,E1 170.095} C_DIS
LIN {X -0.141,Y -368.172,Z 1391.743,A 0.000,B 0.000,C 90.000,E1 169.746} C_DIS
LIN {X 0.089,Y -364.707,Z 1391.738,A 0.000,B 0.000,C 90.000,E1 168.814} C_DIS
LIN {X 0.107,Y -364.105,Z 1391.735,A 0.000,B 0.000,C 90.000,E1 168.342} C_DIS
LIN {X 0.071,Y -364.121,Z 1391.735,A 0.000,B 0.000,C 90.000,E1 168.342} C_DIS
LIN {X -0.083,Y -365.039,Z 1391.733,A 0.000,B 0.000,C 90.000,E1 167.993} C_DIS
LIN {X -0.119,Y -365.061,Z 1391.733,A 0.000,B 0.000,C 90.000,E1 167.993} C_DIS
LIN {X -0.037,Y -367.880,Z 1391.731,A 0.000,B 0.000,C 90.000,E1 167.521} C_DIS
LIN {X -0.153,Y -368.986,Z 1391.730,A 0.000,B 0.000,C 90.000,E1 167.353} C_DIS
LIN {X -0.109,Y -376.310,Z 1391.724,A 0.000,B 0.000,C 90.000,E1 166.408} C_DIS
LIN {X 0.123,Y -383.770,Z 1391.720,A 0.000,B 0.000,C 90.000,E1 165.519} C_DIS
LIN {X -0.016,Y -395.967,Z 1391.713,A 0.000,B 0.000,C 90.000,E1 164.283} C_DIS
LIN {X -0.180,Y -408.392,Z 1391.706,A 0.000,B 0.000,C 90.000,E1 163.142} C_DIS
LIN {X 0.181,Y -435.256,Z 1391.694,A 0.000,B 0.000,C 90.000,E1 160.859} C_DIS
LIN {X 0.135,Y -447.780,Z 1391.688,A 0.000,B 0.000,C 90.000,E1 159.880} C_DIS
LIN {X -0.002,Y -458.710,Z 1391.684,A 0.000,B 0.000,C 90.000,E1 159.028} C_DIS
LIN {X -0.044,Y -466.320,Z 1391.680,A 0.000,B 0.000,C 90.000,E1 158.411} C_DIS
LIN {X -0.048,Y -472.342,Z 1391.677,A 0.000,B 0.000,C 90.000,E1 157.901} C_DIS
LIN {X 0.027,Y -479.633,Z 1391.674,A 0.000,B 0.000,C 90.000,E1 157.230} C_DIS
LIN {X -0.112,Y -489.747,Z 1391.668,A 0.000,B 0.000,C 90.000,E1 156.305} C_DIS
LIN {X 0.082,Y -495.355,Z 1391.665,A 0.000,B 0.000,C 90.000,E1 155.741} C_DIS
LIN {X -0.144,Y -503.551,Z 1391.661,A 0.000,B 0.000,C 90.000,E1 154.921} C_DIS
LIN {X -0.135,Y -510.005,Z 1391.657,A 0.000,B 0.000,C 90.000,E1 154.204} C_DIS
LIN {X 0.101,Y -514.979,Z 1391.653,A 0.000,B 0.000,C 90.000,E1 153.589} C_DIS
LIN {X -0.061,Y -520.847,Z 1391.649,A 0.000,B 0.000,C 90.000,E1 152.871} C_DIS
LIN {X -0.008,Y -525.236,Z 1391.646,A 0.000,B 0.000,C 90.000,E1 152.281} C_DIS
LIN {X -0.013,Y -528.203,Z 1391.644,A 0.000,B 0.000,C 90.000,E1 151.847} C_DIS
LIN {X 0.245,Y -530.946,Z 1391.641,A 0.000,B 0.000,C 90.000,E1 151.385} C_DIS
LIN {X -0.091,Y -534.165,Z 1391.638,A 0.000,B 0.000,C 90.000,E1 150.845} C_DIS
LIN {X 0.066,Y -537.024,Z 1391.635,A 0.000,B 0.000,C 90.000,E1 150.255} C_DIS
LIN {X 0.243,Y -539.455,Z 1391.632,A 0.000,B 0.000,C 90.000,E1 149.665} C_DIS
LIN {X -0.302,Y -542.628,Z 1391.627,A 0.000,B 0.000,C 90.000,E1 148.869} C_DIS
LIN {X -0.094,Y -544.521,Z 1391.624,A 0.000,B 0.000,C 90.000,E1 148.280} C_DIS
LIN {X -0.044,Y -546.211,Z 1391.621,A 0.000,B 0.000,C 90.000,E1 147.709} C_DIS
LIN {X 0.228,Y -548.277,Z 1391.616,A 0.000,B 0.000,C 90.000,E1 146.834} C_DIS
LIN {X 0.062,Y -550.085,Z 1391.611,A 0.000,B 0.000,C 90.000,E1 146.008} C_DIS
LIN {X -0.144,Y -551.154,Z 1391.608,A 0.000,B 0.000,C 90.000,E1 145.468} C_DIS
LIN {X 0.032,Y -552.395,Z 1391.603,A 0.000,B 0.000,C 90.000,E1 144.609} C_DIS
LIN {X -0.097,Y -553.342,Z 1391.599,A 0.000,B 0.000,C 90.000,E1 143.783} C_DIS
LIN {X 0.176,Y -554.365,Z 1391.593,A 0.000,B 0.000,C 90.000,E1 142.637} C_DIS
LIN {X 0.172,Y -555.717,Z 1391.583,A 0.000,B 0.000,C 90.000,E1 140.964} C_DIS
LIN {X 0.037,Y -556.568,Z 1391.577,A 0.000,B 0.000,C 90.000,E1 139.865} C_DIS
LIN {X -0.149,Y -557.206,Z 1391.571,A 0.000,B 0.000,C 90.000,E1 138.771} C_DIS
LIN {X 0.098,Y -557.761,Z 1391.565,A 0.000,B 0.000,C 90.000,E1 137.634} C_DIS
LIN {X 0.168,Y -558.626,Z 1391.552,A 0.000,B 0.000,C 90.000,E1 135.405} C_DIS
LIN {X -0.259,Y -559.183,Z 1391.543,A 0.000,B 0.000,C 90.000,E1 133.785} C_DIS
LIN {X -0.020,Y -559.518,Z 1391.537,A 0.000,B 0.000,C 90.000,E1 132.651} C_DIS
LIN {X -0.001,Y -559.753,Z 1391.528,A 0.000,B 0.000,C 90.000,E1 130.987} C_DIS
LIN {X 0.115,Y -560.150,Z 1391.517,A 0.000,B 0.000,C 90.000,E1 129.036} C_DIS
LIN {X 0.231,Y -560.546,Z 1391.508,A 0.000,B 0.000,C 90.000,E1 127.363} C_DIS
LIN {X 0.017,Y -561.169,Z 1391.499,A 0.000,B 0.000,C 90.000,E1 125.724} C_DIS
LIN {X 0.148,Y -561.849,Z 1391.495,A 0.000,B 0.000,C 90.000,E1 125.025} C_DIS
LIN {X -0.033,Y -562.640,Z 1391.493,A 0.000,B 0.000,C 90.000,E1 124.659} C_DIS
LIN {X -0.075,Y -562.662,Z 1391.493,A 0.000,B 0.000,C 90.000,E1 124.659} C_DIS
LIN {X -0.103,Y -563.837,Z 1391.492,A 0.000,B 0.000,C 90.000,E1 124.485} C_DIS
LIN {X 0.009,Y -564.977,Z 1391.491,A 0.000,B 0.000,C 90.000,E1 124.405} C_DIS
LIN {X -0.037,Y -566.915,Z 1391.491,A 0.000,B 0.000,C 90.000,E1 124.326} C_DIS
LIN {X -0.084,Y -569.914,Z 1391.490,A 0.000,B 0.000,C 90.000,E1 124.246} C_DIS
LIN {X 0.188,Y -575.262,Z 1391.490,A 0.000,B 0.000,C 90.000,E1 124.119} C_DIS
LIN {X -0.002,Y -581.468,Z 1391.489,A 0.000,B 0.000,C 90.000,E1 123.992} C_DIS
LIN {X -0.091,Y -583.926,Z 1391.488,A 0.000,B 0.000,C 90.000,E1 123.913} C_DIS
LIN {X -0.062,Y -586.924,Z 1391.488,A 0.000,B 0.000,C 90.000,E1 123.785} C_DIS
LIN {X -0.253,Y -592.768,Z 1391.486,A 0.000,B 0.000,C 90.000,E1 123.499} C_DIS
LIN {X 0.245,Y -598.518,Z 1391.484,A 0.000,B 0.000,C 90.000,E1 123.086} C_DIS
LIN {X 0.313,Y -601.393,Z 1391.483,A 0.000,B 0.000,C 90.000,E1 122.880} C_DIS
LIN {X 0.144,Y -606.852,Z 1391.480,A 0.000,B 0.000,C 90.000,E1 122.467} C_DIS
LIN {X -0.216,Y -613.525,Z 1391.477,A 0.000,B 0.000,C 90.000,E1 121.926} C_DIS
LIN {X 0.254,Y -619.461,Z 1391.474,A 0.000,B 0.000,C 90.000,E1 121.258} C_DIS
LIN {X 0.236,Y -622.895,Z 1391.472,A 0.000,B 0.000,C 90.000,E1 120.875} C_DIS
LIN {X 0.011,Y -627.092,Z 1391.469,A 0.000,B 0.000,C 90.000,E1 120.384} C_DIS
LIN {X 0.036,Y -630.909,Z 1391.466,A 0.000,B 0.000,C 90.000,E1 119.873} C_DIS
LIN {X 0.092,Y -634.311,Z 1391.463,A 0.000,B 0.000,C 90.000,E1 119.361} C_DIS
LIN {X -0.050,Y -638.136,Z 1391.460,A 0.000,B 0.000,C 90.000,E1 118.743} C_DIS
LIN {X 0.057,Y -640.632,Z 1391.457,A 0.000,B 0.000,C 90.000,E1 118.231} C_DIS
LIN {X 0.119,Y -641.705,Z 1391.456,A 0.000,B 0.000,C 90.000,E1 117.975} C_DIS
LIN {X -0.319,Y -643.484,Z 1391.453,A 0.000,B 0.000,C 90.000,E1 117.513} C_DIS
LIN {X -0.248,Y -644.206,Z 1391.451,A 0.000,B 0.000,C 90.000,E1 117.257} C_DIS
LIN {X -0.174,Y -644.673,Z 1391.450,A 0.000,B 0.000,C 90.000,E1 117.001} C_DIS
LIN {X -0.020,Y -645.268,Z 1391.447,A 0.000,B 0.000,C 90.000,E1 116.488} C_DIS
LIN {X 0.059,Y -645.444,Z 1391.446,A 0.000,B 0.000,C 90.000,E1 116.232} C_DIS
LIN {X 0.220,Y -645.142,Z 1391.443,A 0.000,B 0.000,C 90.000,E1 115.720} C_DIS
LIN {X 0.377,Y -644.537,Z 1391.440,A 0.000,B 0.000,C 90.000,E1 115.207} C_DIS
LIN {X 0.182,Y -644.035,Z 1391.439,A 0.000,B 0.000,C 90.000,E1 114.975} C_DIS
LIN {X -0.251,Y -642.280,Z 1391.436,A 0.000,B 0.000,C 90.000,E1 114.515} C_DIS
LIN {X -0.216,Y -641.561,Z 1391.435,A 0.000,B 0.000,C 90.000,E1 114.387} C_DIS
LIN {X -0.346,Y -637.841,Z 1391.433,A 0.000,B 0.000,C 90.000,E1 113.898} C_DIS
LIN {X -0.316,Y -636.237,Z 1391.432,A 0.000,B 0.000,C 90.000,E1 113.770} C_DIS
LIN {X -0.104,Y -634.396,Z 1391.431,A 0.000,B 0.000,C 90.000,E1 113.643} C_DIS
LIN {X -0.255,Y -630.709,Z 1391.430,A 0.000,B 0.000,C 90.000,E1 113.387} C_DIS
LIN {X 0.292,Y -621.673,Z 1391.428,A 0.000,B 0.000,C 90.000,E1 112.950} C_DIS
LIN {X 0.221,Y -617.750,Z 1391.427,A 0.000,B 0.000,C 90.000,E1 112.823} C_DIS
LIN {X 0.290,Y -606.365,Z 1391.425,A 0.000,B 0.000,C 90.000,E1 112.461} C_DIS
LIN {X 0.255,Y -606.397,Z 1391.425,A 0.000,B 0.000,C 90.000,E1 112.461} C_DIS
LIN {X 0.216,Y -609.113,Z 1391.424,A 0.000,B 0.000,C 90.000,E1 112.206} C_DIS
LIN {X 0.029,Y -615.101,Z 1391.421,A 0.000,B 0.000,C 90.000,E1 111.716} C_DIS
LIN {X 0.260,Y -620.290,Z 1391.418,A 0.000,B 0.000,C 90.000,E1 111.227} C_DIS
END
